% RSLogix 500 project C8014 TOPCOAT B 20170512 CBP.RSS, saved by version 8.30.00.16 %
PROJECT "C8014"    % processor: MicroLogix 1400; MAIN_PROG %

PROGRAM FILES
  LAD 2 "MAIN_PROG"  16 rungs
  LAD 3 "TCB ENTRY"  5 rungs
  LAD 4 "TCB TUNNEL"  44 rungs
  LAD 5 "REWORK"  13 rungs
  LAD 6 "COMMS"  3 rungs
  LAD 7   4 rungs
  LAD 8 "GATE FTA"  12 rungs
  LAD 9 "Z142-145"  23 rungs
  LAD 10 "TO_GLAZE"  15 rungs
  LAD 11 "FROM_GLAZE"  17 rungs
  LAD 12 "TO_BARN"  5 rungs
  LAD 13 "FRM_REPAIR"  5 rungs

DATA FILES
  O0 OUTPUT  9 elements
  I1 INPUT  12 elements
  S2 STATUS  66 elements
  B3 BINARY  40 elements
  T4 TIMER  54 elements
  C5 COUNTER  10 elements
  R6 CONTROL  1 elements
  N7 INTEGER  100 elements
  F8 FLOAT  1 elements
  ST9   21 elements
  RI10   5 elements
  MG11   4 elements

LADDER 2 "MAIN_PROG"
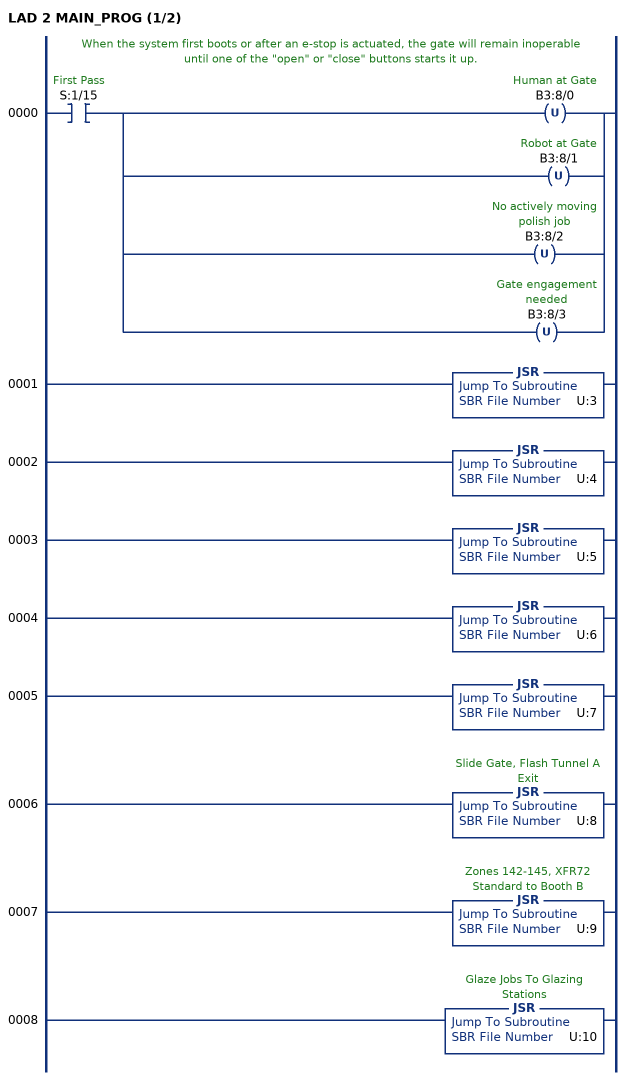
% Rung: 0 %
% When the system first boots or after an e-stop is actuated, the gate will remain inoperable until one of the "open" or "close" buttons starts it up. %
SOR XIC S:1/15 BST OTU B3:8/0 NXB OTU B3:8/1 NXB OTU B3:8/2 NXB OTU B3:8/3 BND EOR
%   S:1/15  "First Pass" %
%   B3:8/0  "Human at Gate" %
%   B3:8/1  "Robot at Gate" %
%   B3:8/2  "No actively moving polish job" %
%   B3:8/3  "Gate engagement needed" %
% Rung: 1 %
SOR JSR U:3 EOR
% Rung: 2 %
SOR JSR U:4 EOR
% Rung: 3 %
SOR JSR U:5 EOR
% Rung: 4 %
SOR JSR U:6 EOR
% Rung: 5 %
SOR JSR U:7 EOR
% Rung: 6 %
SOR JSR U:8 EOR
%   U:8  "Slide Gate, Flash Tunnel A Exit" %
% Rung: 7 %
SOR JSR U:9 EOR
%   U:9  "Zones 142-145, XFR72 Standard to Booth B" %
% Rung: 8 %
SOR JSR U:10 EOR
%   U:10  "Glaze Jobs To Glazing Stations" %

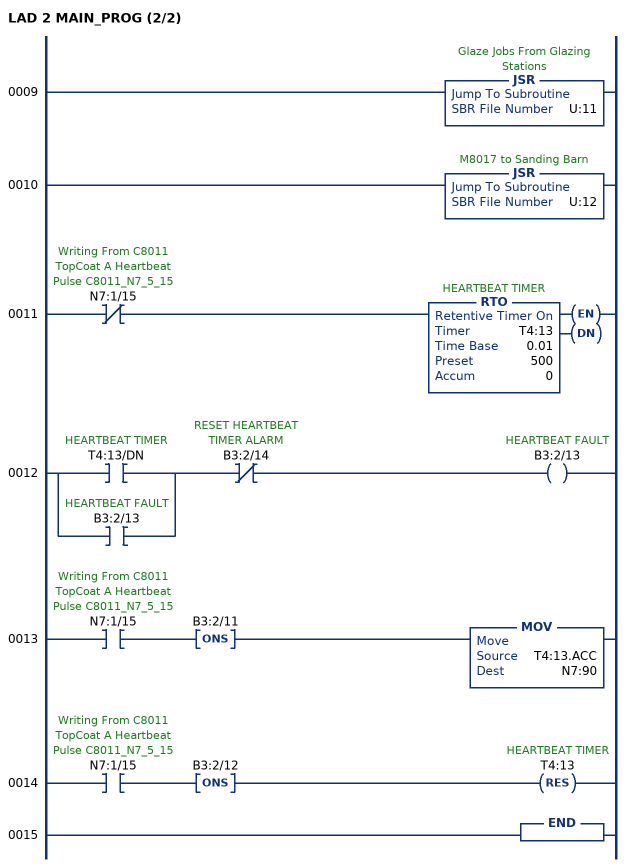
% Rung: 9 %
SOR JSR U:11 EOR
%   U:11  "Glaze Jobs From Glazing Stations" %
% Rung: 10 %
SOR JSR U:12 EOR
%   U:12  "M8017 to Sanding Barn" %
% Rung: 11 %
SOR XIO N7:1/15 RTO T4:13 0.01 500 0 EOR
%   N7:1/15  C8011_N7_5_15  "Writing From C8011 TopCoat A Heartbeat Pulse" %
%   T4:13  "HEARTBEAT TIMER" %
% Rung: 12 %
SOR BST XIC T4:13/DN NXB XIC B3:2/13 BND XIO B3:2/14 OTE B3:2/13 EOR
%   T4:13  "HEARTBEAT TIMER" %
%   B3:2/13  "HEARTBEAT FAULT" %
%   B3:2/14  "RESET HEARTBEAT TIMER ALARM" %
% Rung: 13 %
SOR XIC N7:1/15 ONS B3:2/11 MOV T4:13.ACC N7:90 EOR
%   N7:1/15  C8011_N7_5_15  "Writing From C8011 TopCoat A Heartbeat Pulse" %
%   T4:13  "HEARTBEAT TIMER" %
% Rung: 14 %
SOR XIC N7:1/15 ONS B3:2/12 RES T4:13 EOR
%   N7:1/15  C8011_N7_5_15  "Writing From C8011 TopCoat A Heartbeat Pulse" %
%   T4:13  "HEARTBEAT TIMER" %
% Rung: 15 %
SOR END EOR

LADDER 3 "TCB ENTRY"
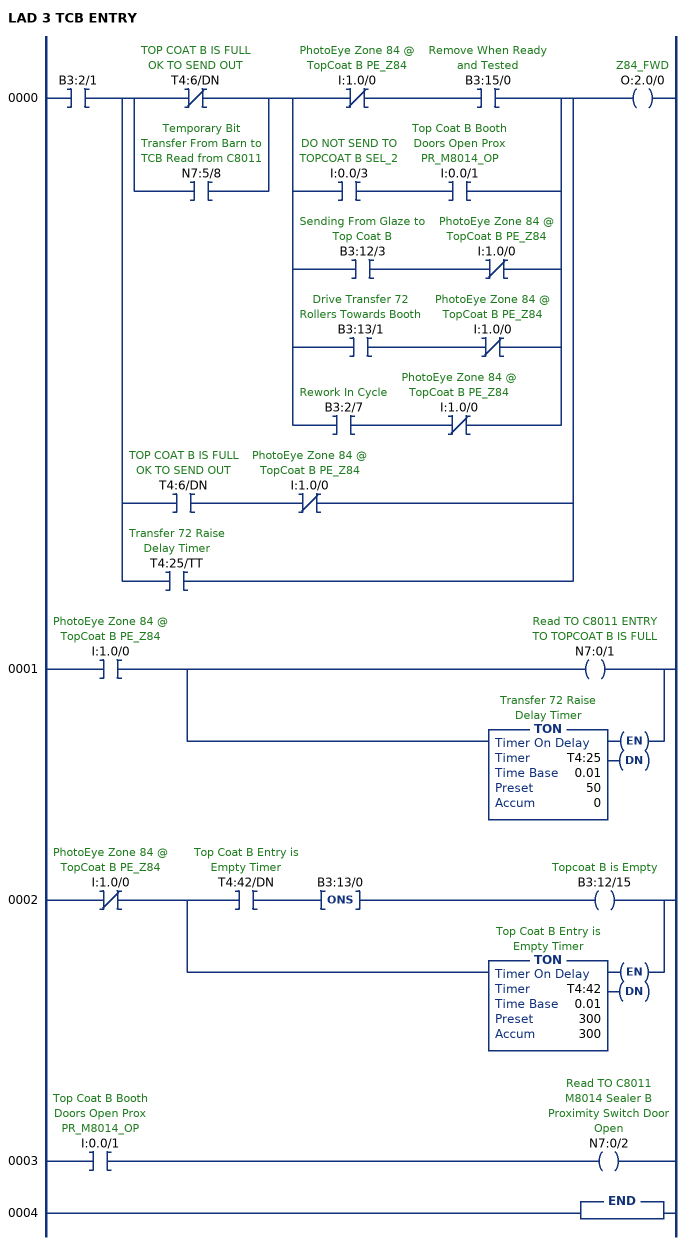
% Rung: 0 %
SOR XIC B3:2/1 BST BST XIO T4:6/DN NXB XIC N7:5/8 BND BST XIO I:1.0/0 XIC B3:15/0 NXB XIC I:0.0/3 XIC I:0.0/1 NXB XIC B3:12/3 XIO I:1.0/0 NXB XIC B3:13/1 XIO I:1.0/0 NXB XIC B3:2/7 XIO I:1.0/0 BND NXB XIC T4:6/DN XIO I:1.0/0 NXB XIC T4:25/TT BND OTE O:2.0/0 EOR
%   T4:6  "TOP COAT B IS FULL OK TO SEND OUT" %
%   N7:5/8  "Temporary Bit Transfer From Barn to TCB Read from C8011" %
%   I:1.0/0  PE_Z84  "PhotoEye Zone 84 @ TopCoat B" %
%   B3:15/0  "Remove When Ready and Tested" %
%   I:0.0/3  SEL_2  "DO NOT SEND TO TOPCOAT B" %
%   I:0.0/1  PR_M8014_OP  "Top Coat B Booth Doors Open Prox" %
%   B3:12/3  "Sending From Glaze to Top Coat B" %
%   B3:13/1  "Drive Transfer 72 Rollers Towards Booth" %
%   B3:2/7  "Rework In Cycle" %
%   T4:25  "Transfer 72 Raise Delay Timer" %
%   O:2.0/0  Z84_FWD %
% Rung: 1 %
SOR XIC I:1.0/0 BST OTE N7:0/1 NXB TON T4:25 0.01 50 0 BND EOR
%   I:1.0/0  PE_Z84  "PhotoEye Zone 84 @ TopCoat B" %
%   N7:0/1  "Read TO C8011 ENTRY TO TOPCOAT B IS FULL" %
%   T4:25  "Transfer 72 Raise Delay Timer" %
% Rung: 2 %
SOR XIO I:1.0/0 BST XIC T4:42/DN ONS B3:13/0 OTE B3:12/15 NXB TON T4:42 0.01 300 300 BND EOR
%   I:1.0/0  PE_Z84  "PhotoEye Zone 84 @ TopCoat B" %
%   T4:42  "Top Coat B Entry is Empty Timer" %
%   B3:12/15  "Topcoat B is Empty" %
% Rung: 3 %
SOR XIC I:0.0/1 OTE N7:0/2 EOR
%   I:0.0/1  PR_M8014_OP  "Top Coat B Booth Doors Open Prox" %
%   N7:0/2  "Read TO C8011 M8014 Sealer B Proximity Switch Door Open" %
% Rung: 4 %
SOR END EOR

LADDER 4 "TCB TUNNEL"
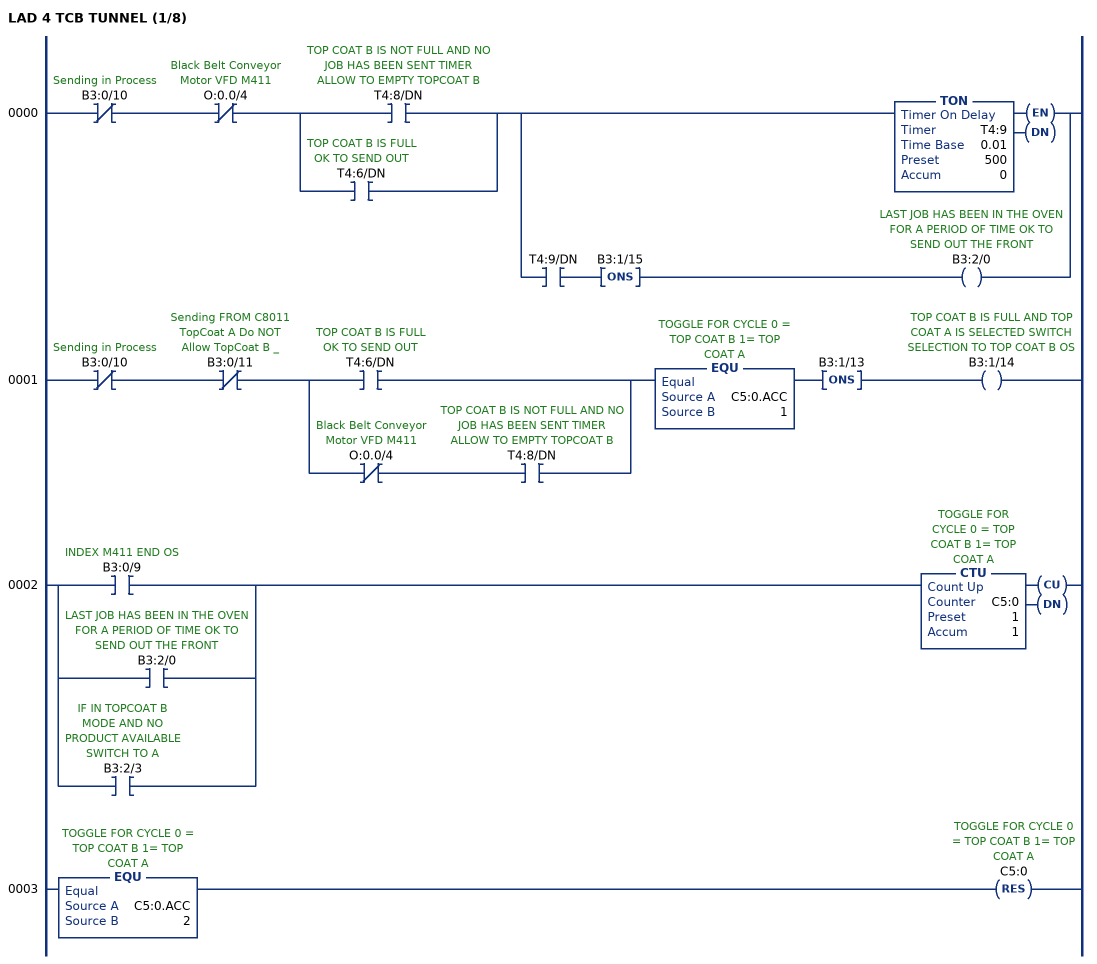
% Rung: 0 %
SOR XIO B3:0/10 XIO O:0.0/4 BST XIC T4:8/DN NXB XIC T4:6/DN BND BST TON T4:9 0.01 500 0 NXB XIC T4:9/DN ONS B3:1/15 OTE B3:2/0 BND EOR
%   B3:0/10  "Sending in Process" %
%   O:0.0/4  M411  "Black Belt Conveyor Motor VFD" %
%   T4:8  "TOP COAT B IS NOT FULL AND NO JOB HAS BEEN SENT TIMER ALLOW TO EMPTY TOPCOAT B" %
%   T4:6  "TOP COAT B IS FULL OK TO SEND OUT" %
%   B3:2/0  "LAST JOB HAS BEEN IN THE OVEN FOR A PERIOD OF TIME OK TO SEND OUT THE FRONT" %
% Rung: 1 %
SOR XIO B3:0/10 XIO B3:0/11 BST XIC T4:6/DN NXB XIO O:0.0/4 XIC T4:8/DN BND EQU C5:0.ACC 1 ONS B3:1/13 OTE B3:1/14 EOR
%   B3:0/10  "Sending in Process" %
%   B3:0/11  _  "Sending FROM C8011 TopCoat A Do NOT Allow TopCoat B" %
%   T4:6  "TOP COAT B IS FULL OK TO SEND OUT" %
%   O:0.0/4  M411  "Black Belt Conveyor Motor VFD" %
%   T4:8  "TOP COAT B IS NOT FULL AND NO JOB HAS BEEN SENT TIMER ALLOW TO EMPTY TOPCOAT B" %
%   C5:0  "TOGGLE FOR CYCLE 0 = TOP COAT B 1= TOP COAT A" %
%   B3:1/14  "TOP COAT B IS FULL AND TOP COAT A IS SELECTED SWITCH SELECTION TO TOP COAT B OS" %
% Rung: 2 %
SOR BST XIC B3:0/9 NXB XIC B3:2/0 NXB XIC B3:2/3 BND CTU C5:0 1 1 EOR
%   B3:0/9  "INDEX M411 END OS" %
%   B3:2/0  "LAST JOB HAS BEEN IN THE OVEN FOR A PERIOD OF TIME OK TO SEND OUT THE FRONT" %
%   B3:2/3  "IF IN TOPCOAT B MODE AND NO PRODUCT AVAILABLE SWITCH TO A" %
%   C5:0  "TOGGLE FOR CYCLE 0 = TOP COAT B 1= TOP COAT A" %
% Rung: 3 %
SOR EQU C5:0.ACC 2 RES C5:0 EOR
%   C5:0  "TOGGLE FOR CYCLE 0 = TOP COAT B 1= TOP COAT A" %

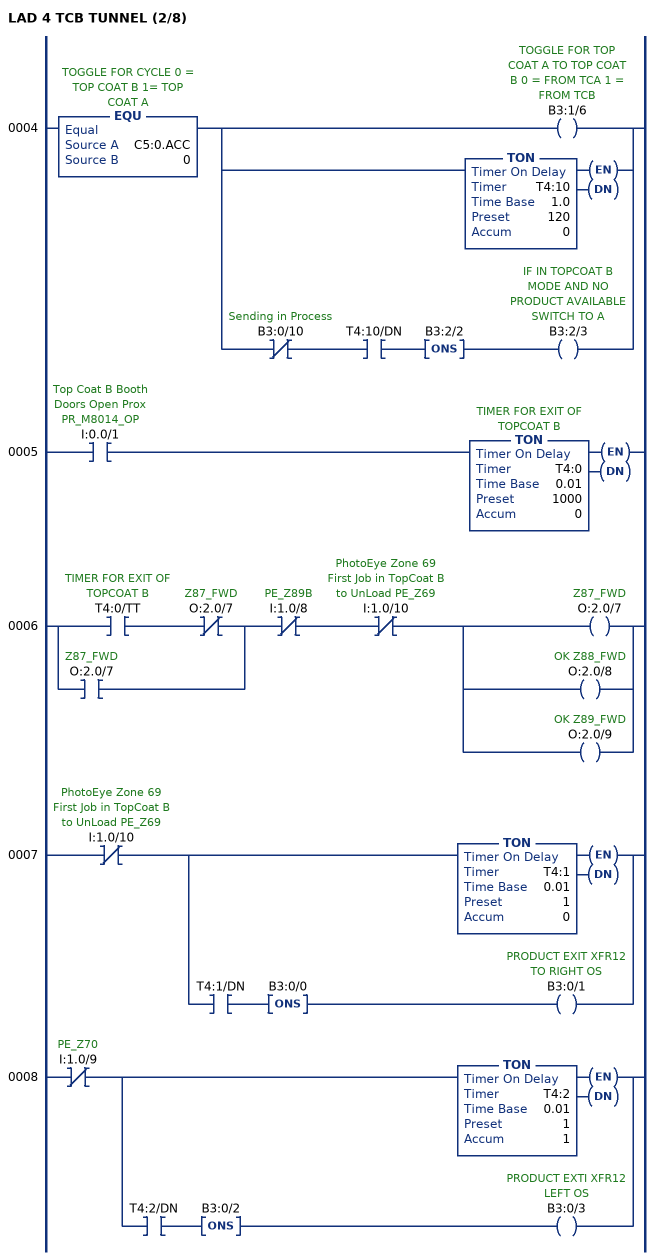
% Rung: 4 %
SOR EQU C5:0.ACC 0 BST OTE B3:1/6 NXB TON T4:10 1.0 120 0 NXB XIO B3:0/10 XIC T4:10/DN ONS B3:2/2 OTE B3:2/3 BND EOR
%   C5:0  "TOGGLE FOR CYCLE 0 = TOP COAT B 1= TOP COAT A" %
%   B3:1/6  "TOGGLE FOR TOP COAT A TO TOP COAT B 0 = FROM TCA 1 = FROM TCB" %
%   B3:0/10  "Sending in Process" %
%   B3:2/3  "IF IN TOPCOAT B MODE AND NO PRODUCT AVAILABLE SWITCH TO A" %
% Rung: 5 %
SOR XIC I:0.0/1 TON T4:0 0.01 1000 0 EOR
%   I:0.0/1  PR_M8014_OP  "Top Coat B Booth Doors Open Prox" %
%   T4:0  "TIMER FOR EXIT OF TOPCOAT B" %
% Rung: 6 %
SOR BST XIC T4:0/TT XIO O:2.0/7 NXB XIC O:2.0/7 BND XIO I:1.0/8 XIO I:1.0/10 BST OTE O:2.0/7 NXB OTE O:2.0/8 NXB OTE O:2.0/9 BND EOR
%   T4:0  "TIMER FOR EXIT OF TOPCOAT B" %
%   O:2.0/7  Z87_FWD %
%   I:1.0/8  PE_Z89B %
%   I:1.0/10  PE_Z69  "PhotoEye Zone 69 First Job in TopCoat B to UnLoad" %
%   O:2.0/8  Z88_FWD  "OK" %
%   O:2.0/9  Z89_FWD  "OK" %
% Rung: 7 %
SOR XIO I:1.0/10 BST TON T4:1 0.01 1 0 NXB XIC T4:1/DN ONS B3:0/0 OTE B3:0/1 BND EOR
%   I:1.0/10  PE_Z69  "PhotoEye Zone 69 First Job in TopCoat B to UnLoad" %
%   B3:0/1  "PRODUCT EXIT XFR12 TO RIGHT OS" %
% Rung: 8 %
SOR XIO I:1.0/9 BST TON T4:2 0.01 1 1 NXB XIC T4:2/DN ONS B3:0/2 OTE B3:0/3 BND EOR
%   I:1.0/9  PE_Z70 %
%   B3:0/3  "PRODUCT EXTI XFR12 LEFT OS" %

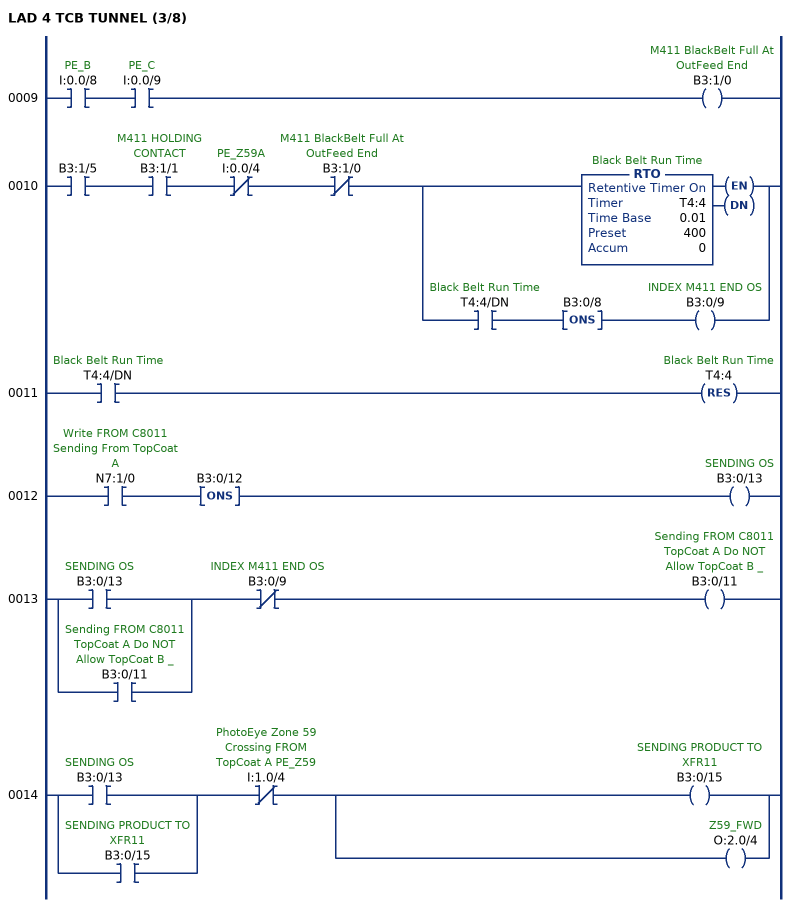
% Rung: 9 %
SOR XIC I:0.0/8 XIC I:0.0/9 OTE B3:1/0 EOR
%   I:0.0/8  PE_B %
%   I:0.0/9  PE_C %
%   B3:1/0  "M411 BlackBelt Full At OutFeed End" %
% Rung: 10 %
SOR XIC B3:1/5 XIC B3:1/1 XIO I:0.0/4 XIO B3:1/0 BST RTO T4:4 0.01 400 0 NXB XIC T4:4/DN ONS B3:0/8 OTE B3:0/9 BND EOR
%   B3:1/1  "M411 HOLDING CONTACT" %
%   I:0.0/4  PE_Z59A %
%   B3:1/0  "M411 BlackBelt Full At OutFeed End" %
%   T4:4  "Black Belt Run Time" %
%   B3:0/9  "INDEX M411 END OS" %
% Rung: 11 %
SOR XIC T4:4/DN RES T4:4 EOR
%   T4:4  "Black Belt Run Time" %
% Rung: 12 %
SOR XIC N7:1/0 ONS B3:0/12 OTE B3:0/13 EOR
%   N7:1/0  "Write FROM C8011 Sending From TopCoat A" %
%   B3:0/13  "SENDING OS" %
% Rung: 13 %
SOR BST XIC B3:0/13 NXB XIC B3:0/11 BND XIO B3:0/9 OTE B3:0/11 EOR
%   B3:0/13  "SENDING OS" %
%   B3:0/11  _  "Sending FROM C8011 TopCoat A Do NOT Allow TopCoat B" %
%   B3:0/9  "INDEX M411 END OS" %
% Rung: 14 %
SOR BST XIC B3:0/13 NXB XIC B3:0/15 BND XIO I:1.0/4 BST OTE B3:0/15 NXB OTE O:2.0/4 BND EOR
%   B3:0/13  "SENDING OS" %
%   B3:0/15  "SENDING PRODUCT TO XFR11" %
%   I:1.0/4  PE_Z59  "PhotoEye Zone 59 Crossing FROM TopCoat A" %
%   O:2.0/4  Z59_FWD %

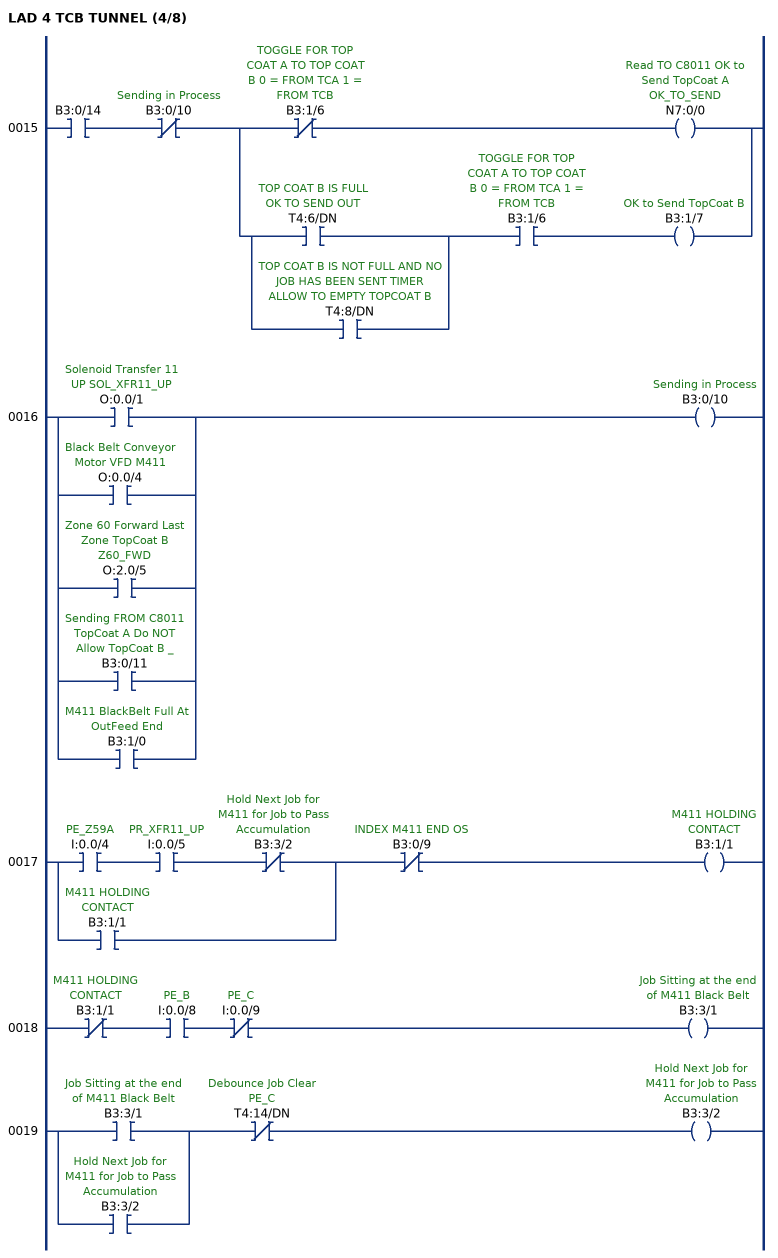
% Rung: 15 %
SOR XIC B3:0/14 XIO B3:0/10 BST XIO B3:1/6 OTE N7:0/0 NXB BST XIC T4:6/DN NXB XIC T4:8/DN BND XIC B3:1/6 OTE B3:1/7 BND EOR
%   B3:0/10  "Sending in Process" %
%   B3:1/6  "TOGGLE FOR TOP COAT A TO TOP COAT B 0 = FROM TCA 1 = FROM TCB" %
%   N7:0/0  OK_TO_SEND  "Read TO C8011 OK to Send TopCoat A" %
%   T4:6  "TOP COAT B IS FULL OK TO SEND OUT" %
%   T4:8  "TOP COAT B IS NOT FULL AND NO JOB HAS BEEN SENT TIMER ALLOW TO EMPTY TOPCOAT B" %
%   B3:1/7  "OK to Send TopCoat B" %
% Rung: 16 %
SOR BST XIC O:0.0/1 NXB XIC O:0.0/4 NXB XIC O:2.0/5 NXB XIC B3:0/11 NXB XIC B3:1/0 BND OTE B3:0/10 EOR
%   O:0.0/1  SOL_XFR11_UP  "Solenoid Transfer 11 UP" %
%   O:0.0/4  M411  "Black Belt Conveyor Motor VFD" %
%   O:2.0/5  Z60_FWD  "Zone 60 Forward Last Zone TopCoat B" %
%   B3:0/11  _  "Sending FROM C8011 TopCoat A Do NOT Allow TopCoat B" %
%   B3:1/0  "M411 BlackBelt Full At OutFeed End" %
%   B3:0/10  "Sending in Process" %
% Rung: 17 %
SOR BST XIC I:0.0/4 XIC I:0.0/5 XIO B3:3/2 NXB XIC B3:1/1 BND XIO B3:0/9 OTE B3:1/1 EOR
%   I:0.0/4  PE_Z59A %
%   I:0.0/5  PR_XFR11_UP %
%   B3:3/2  "Hold Next Job for M411 for Job to Pass Accumulation" %
%   B3:1/1  "M411 HOLDING CONTACT" %
%   B3:0/9  "INDEX M411 END OS" %
% Rung: 18 %
SOR XIO B3:1/1 XIC I:0.0/8 XIO I:0.0/9 OTE B3:3/1 EOR
%   B3:1/1  "M411 HOLDING CONTACT" %
%   I:0.0/8  PE_B %
%   I:0.0/9  PE_C %
%   B3:3/1  "Job Sitting at the end of M411 Black Belt" %
% Rung: 19 %
SOR BST XIC B3:3/1 NXB XIC B3:3/2 BND XIO T4:14/DN OTE B3:3/2 EOR
%   B3:3/1  "Job Sitting at the end of M411 Black Belt" %
%   B3:3/2  "Hold Next Job for M411 for Job to Pass Accumulation" %
%   T4:14  "Debounce Job Clear PE_C" %

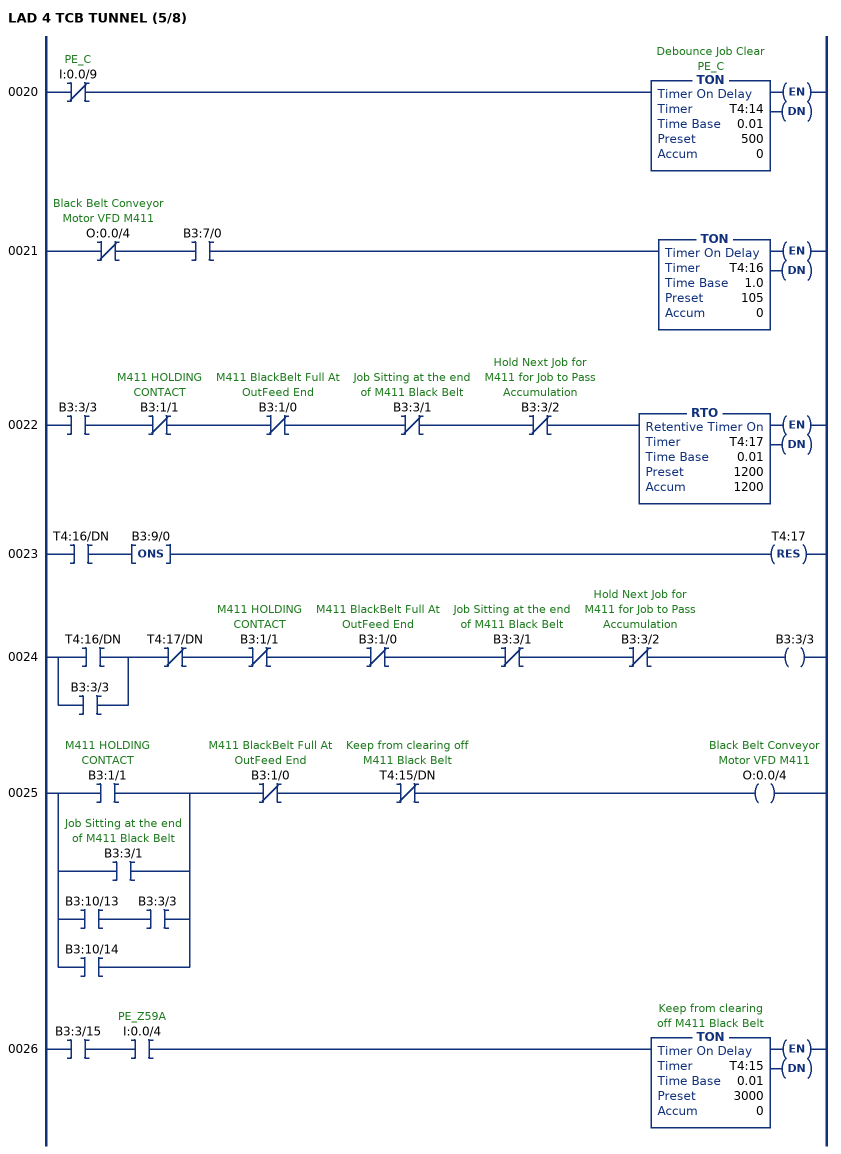
% Rung: 20 %
SOR XIO I:0.0/9 TON T4:14 0.01 500 0 EOR
%   I:0.0/9  PE_C %
%   T4:14  "Debounce Job Clear PE_C" %
% Rung: 21 %
SOR XIO O:0.0/4 XIC B3:7/0 TON T4:16 1.0 105 0 EOR
%   O:0.0/4  M411  "Black Belt Conveyor Motor VFD" %
% Rung: 22 %
SOR XIC B3:3/3 XIO B3:1/1 XIO B3:1/0 XIO B3:3/1 XIO B3:3/2 RTO T4:17 0.01 1200 1200 EOR
%   B3:1/1  "M411 HOLDING CONTACT" %
%   B3:1/0  "M411 BlackBelt Full At OutFeed End" %
%   B3:3/1  "Job Sitting at the end of M411 Black Belt" %
%   B3:3/2  "Hold Next Job for M411 for Job to Pass Accumulation" %
% Rung: 23 %
SOR XIC T4:16/DN ONS B3:9/0 RES T4:17 EOR
% Rung: 24 %
SOR BST XIC T4:16/DN NXB XIC B3:3/3 BND XIO T4:17/DN XIO B3:1/1 XIO B3:1/0 XIO B3:3/1 XIO B3:3/2 OTE B3:3/3 EOR
%   B3:1/1  "M411 HOLDING CONTACT" %
%   B3:1/0  "M411 BlackBelt Full At OutFeed End" %
%   B3:3/1  "Job Sitting at the end of M411 Black Belt" %
%   B3:3/2  "Hold Next Job for M411 for Job to Pass Accumulation" %
% Rung: 25 %
SOR BST XIC B3:1/1 NXB XIC B3:3/1 NXB XIC B3:10/13 XIC B3:3/3 NXB XIC B3:10/14 BND XIO B3:1/0 XIO T4:15/DN OTE O:0.0/4 EOR
%   B3:1/1  "M411 HOLDING CONTACT" %
%   B3:3/1  "Job Sitting at the end of M411 Black Belt" %
%   B3:1/0  "M411 BlackBelt Full At OutFeed End" %
%   T4:15  "Keep from clearing off M411 Black Belt" %
%   O:0.0/4  M411  "Black Belt Conveyor Motor VFD" %
% Rung: 26 %
SOR XIC B3:3/15 XIC I:0.0/4 TON T4:15 0.01 3000 0 EOR
%   I:0.0/4  PE_Z59A %
%   T4:15  "Keep from clearing off M411 Black Belt" %

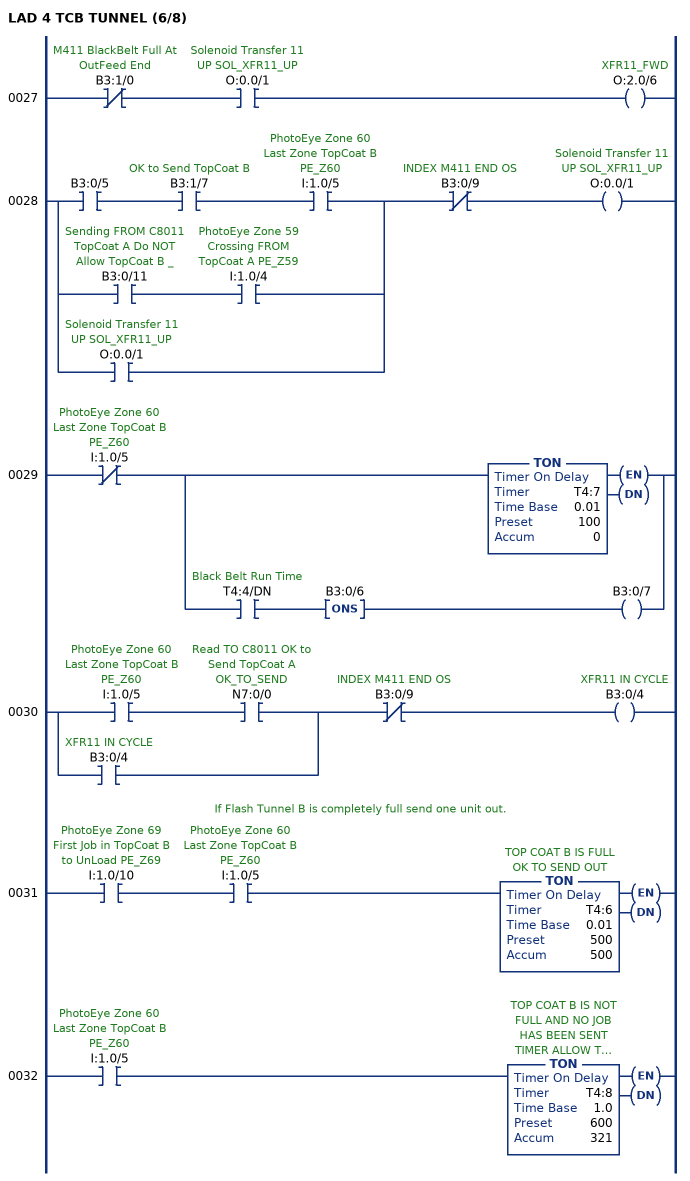
% Rung: 27 %
SOR XIO B3:1/0 XIC O:0.0/1 OTE O:2.0/6 EOR
%   B3:1/0  "M411 BlackBelt Full At OutFeed End" %
%   O:0.0/1  SOL_XFR11_UP  "Solenoid Transfer 11 UP" %
%   O:2.0/6  XFR11_FWD %
% Rung: 28 %
SOR BST BST XIC B3:0/5 XIC B3:1/7 XIC I:1.0/5 NXB XIC B3:0/11 XIC I:1.0/4 BND NXB XIC O:0.0/1 BND XIO B3:0/9 OTE O:0.0/1 EOR
%   B3:1/7  "OK to Send TopCoat B" %
%   I:1.0/5  PE_Z60  "PhotoEye Zone 60 Last Zone TopCoat B" %
%   B3:0/11  _  "Sending FROM C8011 TopCoat A Do NOT Allow TopCoat B" %
%   I:1.0/4  PE_Z59  "PhotoEye Zone 59 Crossing FROM TopCoat A" %
%   O:0.0/1  SOL_XFR11_UP  "Solenoid Transfer 11 UP" %
%   B3:0/9  "INDEX M411 END OS" %
% Rung: 29 %
SOR XIO I:1.0/5 BST TON T4:7 0.01 100 0 NXB XIC T4:4/DN ONS B3:0/6 OTE B3:0/7 BND EOR
%   I:1.0/5  PE_Z60  "PhotoEye Zone 60 Last Zone TopCoat B" %
%   T4:4  "Black Belt Run Time" %
% Rung: 30 %
SOR BST XIC I:1.0/5 XIC N7:0/0 NXB XIC B3:0/4 BND XIO B3:0/9 OTE B3:0/4 EOR
%   I:1.0/5  PE_Z60  "PhotoEye Zone 60 Last Zone TopCoat B" %
%   N7:0/0  OK_TO_SEND  "Read TO C8011 OK to Send TopCoat A" %
%   B3:0/4  "XFR11 IN CYCLE" %
%   B3:0/9  "INDEX M411 END OS" %
% Rung: 31 %
% If Flash Tunnel B is completely full send one unit out. %
SOR XIC I:1.0/10 XIC I:1.0/5 TON T4:6 0.01 500 500 EOR
%   I:1.0/10  PE_Z69  "PhotoEye Zone 69 First Job in TopCoat B to UnLoad" %
%   I:1.0/5  PE_Z60  "PhotoEye Zone 60 Last Zone TopCoat B" %
%   T4:6  "TOP COAT B IS FULL OK TO SEND OUT" %
% Rung: 32 %
SOR XIC I:1.0/5 TON T4:8 1.0 600 321 EOR
%   I:1.0/5  PE_Z60  "PhotoEye Zone 60 Last Zone TopCoat B" %
%   T4:8  "TOP COAT B IS NOT FULL AND NO JOB HAS BEEN SENT TIMER ALLOW TO EMPTY TOPCOAT B" %

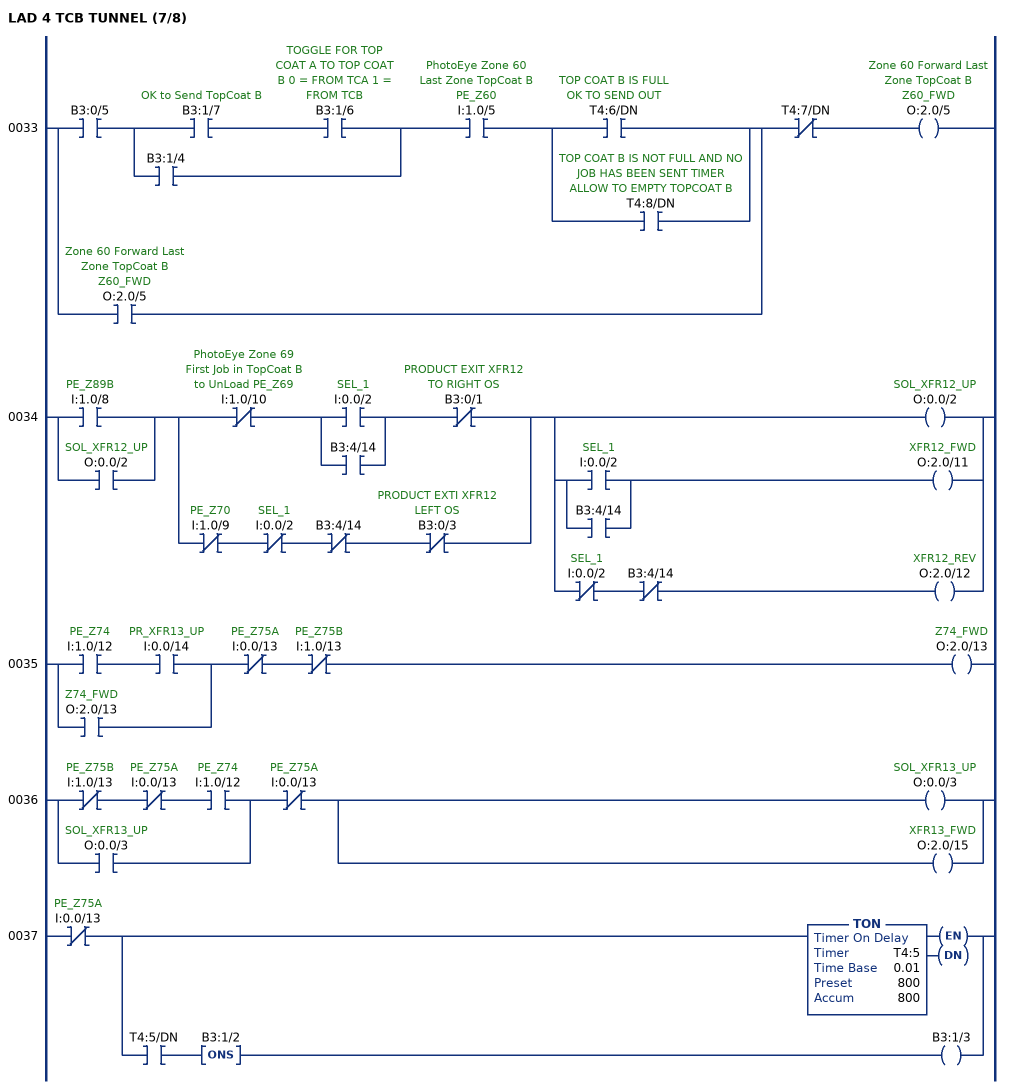
% Rung: 33 %
SOR BST XIC B3:0/5 BST XIC B3:1/7 XIC B3:1/6 NXB XIC B3:1/4 BND XIC I:1.0/5 BST XIC T4:6/DN NXB XIC T4:8/DN BND NXB XIC O:2.0/5 BND XIO T4:7/DN OTE O:2.0/5 EOR
%   B3:1/7  "OK to Send TopCoat B" %
%   B3:1/6  "TOGGLE FOR TOP COAT A TO TOP COAT B 0 = FROM TCA 1 = FROM TCB" %
%   I:1.0/5  PE_Z60  "PhotoEye Zone 60 Last Zone TopCoat B" %
%   T4:6  "TOP COAT B IS FULL OK TO SEND OUT" %
%   T4:8  "TOP COAT B IS NOT FULL AND NO JOB HAS BEEN SENT TIMER ALLOW TO EMPTY TOPCOAT B" %
%   O:2.0/5  Z60_FWD  "Zone 60 Forward Last Zone TopCoat B" %
% Rung: 34 %
SOR BST XIC I:1.0/8 NXB XIC O:0.0/2 BND BST XIO I:1.0/10 BST XIC I:0.0/2 NXB XIC B3:4/14 BND XIO B3:0/1 NXB XIO I:1.0/9 XIO I:0.0/2 XIO B3:4/14 XIO B3:0/3 BND BST OTE O:0.0/2 NXB BST XIC I:0.0/2 NXB XIC B3:4/14 BND OTE O:2.0/11 NXB XIO I:0.0/2 XIO B3:4/14 OTE O:2.0/12 BND EOR
%   I:1.0/8  PE_Z89B %
%   O:0.0/2  SOL_XFR12_UP %
%   I:1.0/10  PE_Z69  "PhotoEye Zone 69 First Job in TopCoat B to UnLoad" %
%   I:0.0/2  SEL_1 %
%   B3:0/1  "PRODUCT EXIT XFR12 TO RIGHT OS" %
%   I:1.0/9  PE_Z70 %
%   B3:0/3  "PRODUCT EXTI XFR12 LEFT OS" %
%   O:2.0/11  XFR12_FWD %
%   O:2.0/12  XFR12_REV %
% Rung: 35 %
SOR BST XIC I:1.0/12 XIC I:0.0/14 NXB XIC O:2.0/13 BND XIO I:0.0/13 XIO I:1.0/13 OTE O:2.0/13 EOR
%   I:1.0/12  PE_Z74 %
%   I:0.0/14  PR_XFR13_UP %
%   O:2.0/13  Z74_FWD %
%   I:0.0/13  PE_Z75A %
%   I:1.0/13  PE_Z75B %
% Rung: 36 %
SOR BST XIO I:1.0/13 XIO I:0.0/13 XIC I:1.0/12 NXB XIC O:0.0/3 BND XIO I:0.0/13 BST OTE O:0.0/3 NXB OTE O:2.0/15 BND EOR
%   I:1.0/13  PE_Z75B %
%   I:0.0/13  PE_Z75A %
%   I:1.0/12  PE_Z74 %
%   O:0.0/3  SOL_XFR13_UP %
%   O:2.0/15  XFR13_FWD %
% Rung: 37 %
SOR XIO I:0.0/13 BST TON T4:5 0.01 800 800 NXB XIC T4:5/DN ONS B3:1/2 OTE B3:1/3 BND EOR
%   I:0.0/13  PE_Z75A %

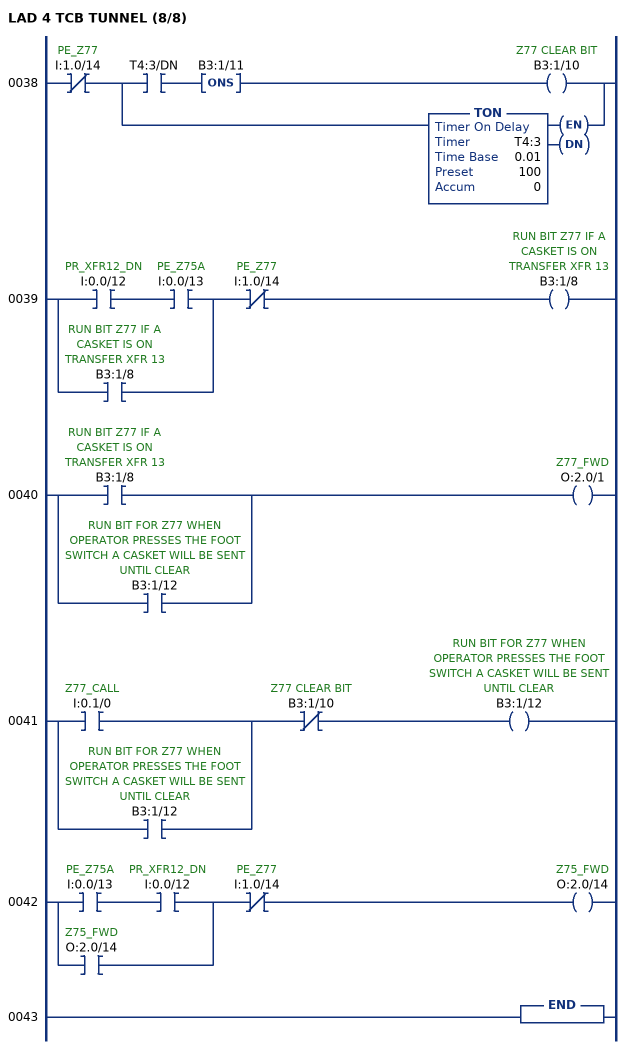
% Rung: 38 %
SOR XIO I:1.0/14 BST XIC T4:3/DN ONS B3:1/11 OTE B3:1/10 NXB TON T4:3 0.01 100 0 BND EOR
%   I:1.0/14  PE_Z77 %
%   B3:1/10  "Z77 CLEAR BIT" %
% Rung: 39 %
SOR BST XIC I:0.0/12 XIC I:0.0/13 NXB XIC B3:1/8 BND XIO I:1.0/14 OTE B3:1/8 EOR
%   I:0.0/12  PR_XFR12_DN %
%   I:0.0/13  PE_Z75A %
%   B3:1/8  "RUN BIT Z77 IF A CASKET IS ON TRANSFER XFR 13" %
%   I:1.0/14  PE_Z77 %
% Rung: 40 %
SOR BST XIC B3:1/8 NXB XIC B3:1/12 BND OTE O:2.0/1 EOR
%   B3:1/8  "RUN BIT Z77 IF A CASKET IS ON TRANSFER XFR 13" %
%   B3:1/12  "RUN BIT FOR Z77 WHEN OPERATOR PRESSES THE FOOT SWITCH A CASKET WILL BE SENT UNTIL CLEAR" %
%   O:2.0/1  Z77_FWD %
% Rung: 41 %
SOR BST XIC I:0.1/0 NXB XIC B3:1/12 BND XIO B3:1/10 OTE B3:1/12 EOR
%   I:0.1/0  Z77_CALL %
%   B3:1/12  "RUN BIT FOR Z77 WHEN OPERATOR PRESSES THE FOOT SWITCH A CASKET WILL BE SENT UNTIL CLEAR" %
%   B3:1/10  "Z77 CLEAR BIT" %
% Rung: 42 %
SOR BST XIC I:0.0/13 XIC I:0.0/12 NXB XIC O:2.0/14 BND XIO I:1.0/14 OTE O:2.0/14 EOR
%   I:0.0/13  PE_Z75A %
%   I:0.0/12  PR_XFR12_DN %
%   O:2.0/14  Z75_FWD %
%   I:1.0/14  PE_Z77 %
% Rung: 43 %
SOR END EOR

LADDER 5 "REWORK"
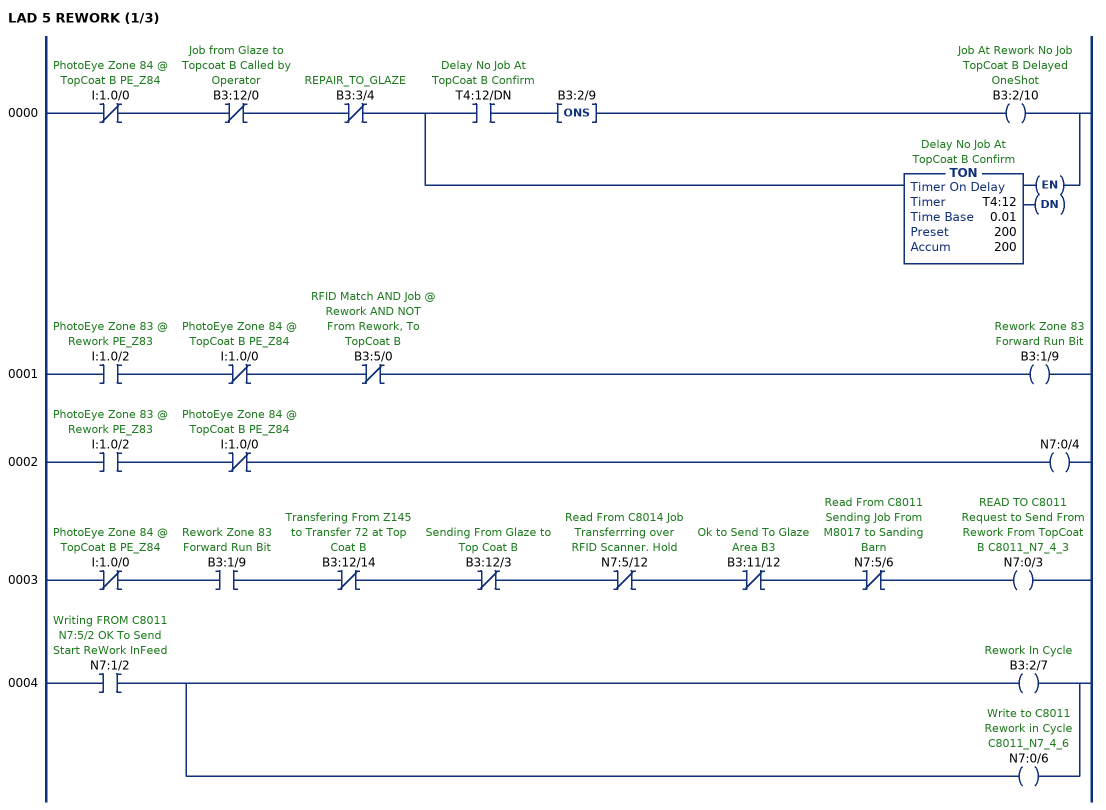
% Rung: 0 %
SOR XIO I:1.0/0 XIO B3:12/0 XIO B3:3/4 BST XIC T4:12/DN ONS B3:2/9 OTE B3:2/10 NXB TON T4:12 0.01 200 200 BND EOR
%   I:1.0/0  PE_Z84  "PhotoEye Zone 84 @ TopCoat B" %
%   B3:12/0  "Job from Glaze to Topcoat B Called by Operator" %
%   B3:3/4  REPAIR_TO_GLAZE %
%   T4:12  "Delay No Job At TopCoat B Confirm" %
%   B3:2/10  "Job At Rework No Job TopCoat B Delayed OneShot" %
% Rung: 1 %
SOR XIC I:1.0/2 XIO I:1.0/0 XIO B3:5/0 OTE B3:1/9 EOR
%   I:1.0/2  PE_Z83  "PhotoEye Zone 83 @ Rework" %
%   I:1.0/0  PE_Z84  "PhotoEye Zone 84 @ TopCoat B" %
%   B3:5/0  "RFID Match AND Job @ Rework AND NOT From Rework, To TopCoat B" %
%   B3:1/9  "Rework Zone 83 Forward Run Bit" %
% Rung: 2 %
SOR XIC I:1.0/2 XIO I:1.0/0 OTE N7:0/4 EOR
%   I:1.0/2  PE_Z83  "PhotoEye Zone 83 @ Rework" %
%   I:1.0/0  PE_Z84  "PhotoEye Zone 84 @ TopCoat B" %
% Rung: 3 %
SOR XIO I:1.0/0 XIC B3:1/9 XIO B3:12/14 XIO B3:12/3 XIO N7:5/12 XIO B3:11/12 XIO N7:5/6 OTE N7:0/3 EOR
%   I:1.0/0  PE_Z84  "PhotoEye Zone 84 @ TopCoat B" %
%   B3:1/9  "Rework Zone 83 Forward Run Bit" %
%   B3:12/14  "Transfering From Z145 to Transfer 72 at Top Coat B" %
%   B3:12/3  "Sending From Glaze to Top Coat B" %
%   N7:5/12  "Read From C8014 Job Transferrring over RFID Scanner. Hold" %
%   B3:11/12  B3  "Ok to Send To Glaze Area" %
%   N7:5/6  "Read From C8011 Sending Job From M8017 to Sanding Barn" %
%   N7:0/3  C8011_N7_4_3  "READ TO C8011 Request to Send From Rework From TopCoat B" %
% Rung: 4 %
SOR XIC N7:1/2 BST OTE B3:2/7 NXB OTE N7:0/6 BND EOR
%   N7:1/2  "Writing FROM C8011 N7:5/2 OK To Send Start ReWork InFeed" %
%   B3:2/7  "Rework In Cycle" %
%   N7:0/6  C8011_N7_4_6  "Write to C8011 Rework in Cycle" %

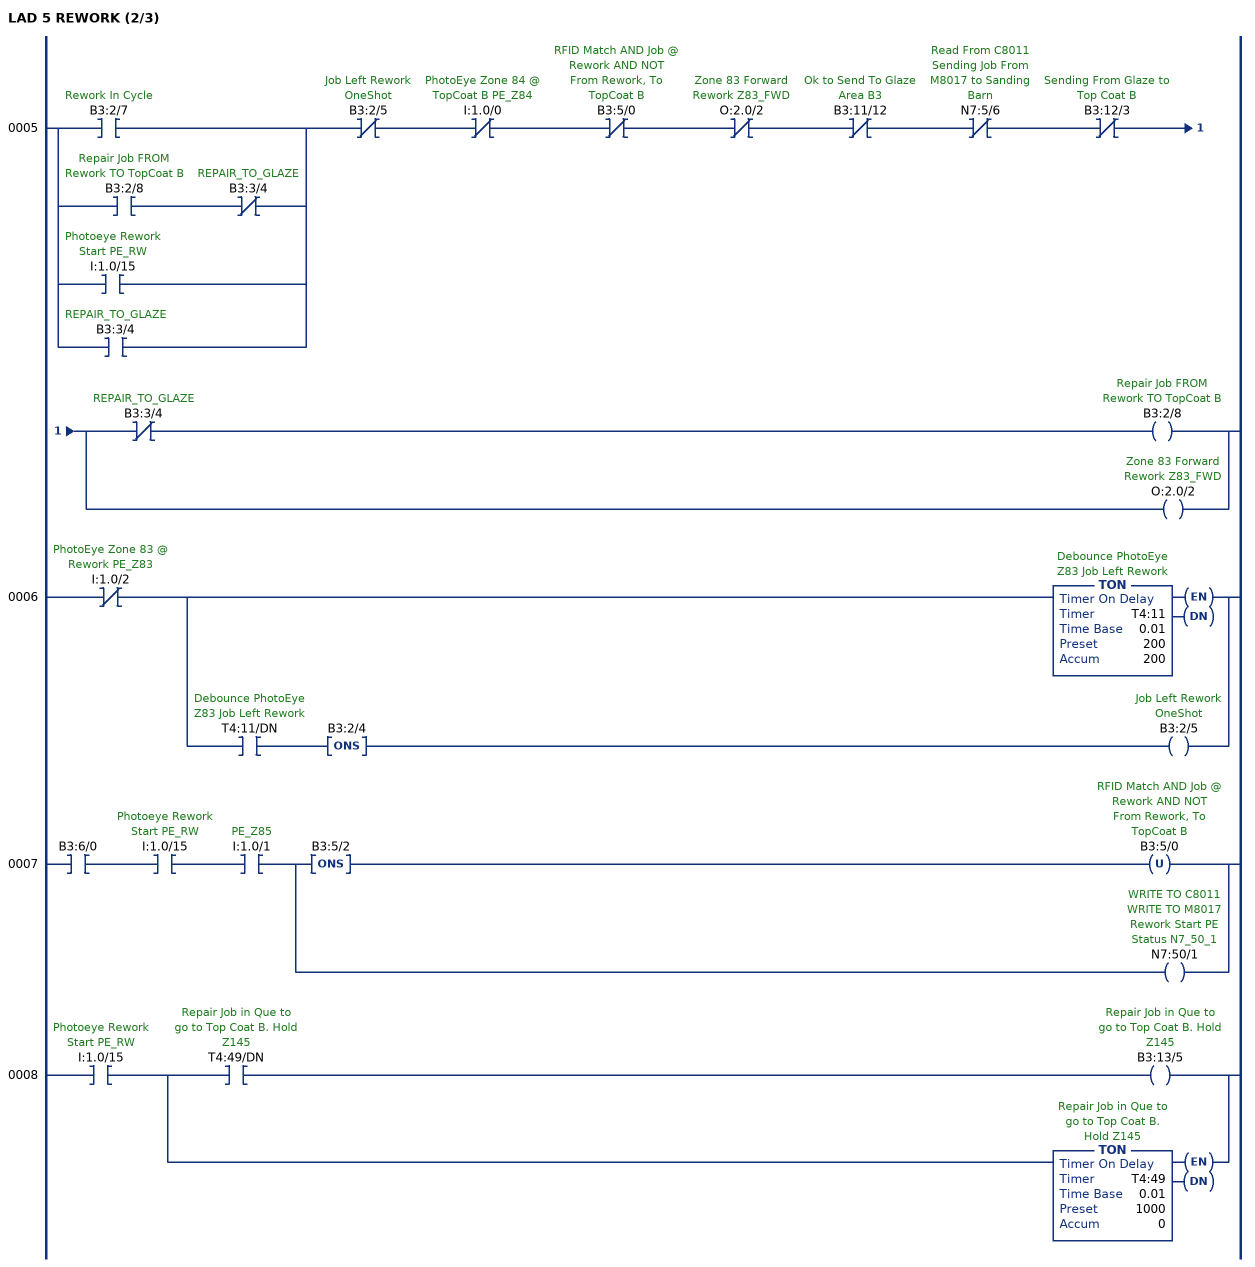
% Rung: 5 %
SOR BST XIC B3:2/7 NXB XIC B3:2/8 XIO B3:3/4 NXB XIC I:1.0/15 NXB XIC B3:3/4 BND XIO B3:2/5 XIO I:1.0/0 XIO B3:5/0 XIO O:2.0/2 XIO B3:11/12 XIO N7:5/6 XIO B3:12/3 BST XIO B3:3/4 OTE B3:2/8 NXB OTE O:2.0/2 BND EOR
%   B3:2/7  "Rework In Cycle" %
%   B3:2/8  "Repair Job FROM Rework TO TopCoat B" %
%   B3:3/4  REPAIR_TO_GLAZE %
%   I:1.0/15  PE_RW  "Photoeye Rework Start" %
%   B3:2/5  "Job Left Rework OneShot" %
%   I:1.0/0  PE_Z84  "PhotoEye Zone 84 @ TopCoat B" %
%   B3:5/0  "RFID Match AND Job @ Rework AND NOT From Rework, To TopCoat B" %
%   O:2.0/2  Z83_FWD  "Zone 83 Forward Rework" %
%   B3:11/12  B3  "Ok to Send To Glaze Area" %
%   N7:5/6  "Read From C8011 Sending Job From M8017 to Sanding Barn" %
%   B3:12/3  "Sending From Glaze to Top Coat B" %
% Rung: 6 %
SOR XIO I:1.0/2 BST TON T4:11 0.01 200 200 NXB XIC T4:11/DN ONS B3:2/4 OTE B3:2/5 BND EOR
%   I:1.0/2  PE_Z83  "PhotoEye Zone 83 @ Rework" %
%   T4:11  "Debounce PhotoEye Z83 Job Left Rework" %
%   B3:2/5  "Job Left Rework OneShot" %
% Rung: 7 %
SOR XIC B3:6/0 XIC I:1.0/15 XIC I:1.0/1 BST ONS B3:5/2 OTU B3:5/0 NXB OTE N7:50/1 BND EOR
%   I:1.0/15  PE_RW  "Photoeye Rework Start" %
%   I:1.0/1  PE_Z85 %
%   B3:5/0  "RFID Match AND Job @ Rework AND NOT From Rework, To TopCoat B" %
%   N7:50/1  N7_50_1  "WRITE TO C8011 WRITE TO M8017 Rework Start PE Status" %
% Rung: 8 %
SOR XIC I:1.0/15 BST XIC T4:49/DN OTE B3:13/5 NXB TON T4:49 0.01 1000 0 BND EOR
%   I:1.0/15  PE_RW  "Photoeye Rework Start" %
%   T4:49  "Repair Job in Que to go to Top Coat B. Hold Z145" %
%   B3:13/5  "Repair Job in Que to go to Top Coat B. Hold Z145" %

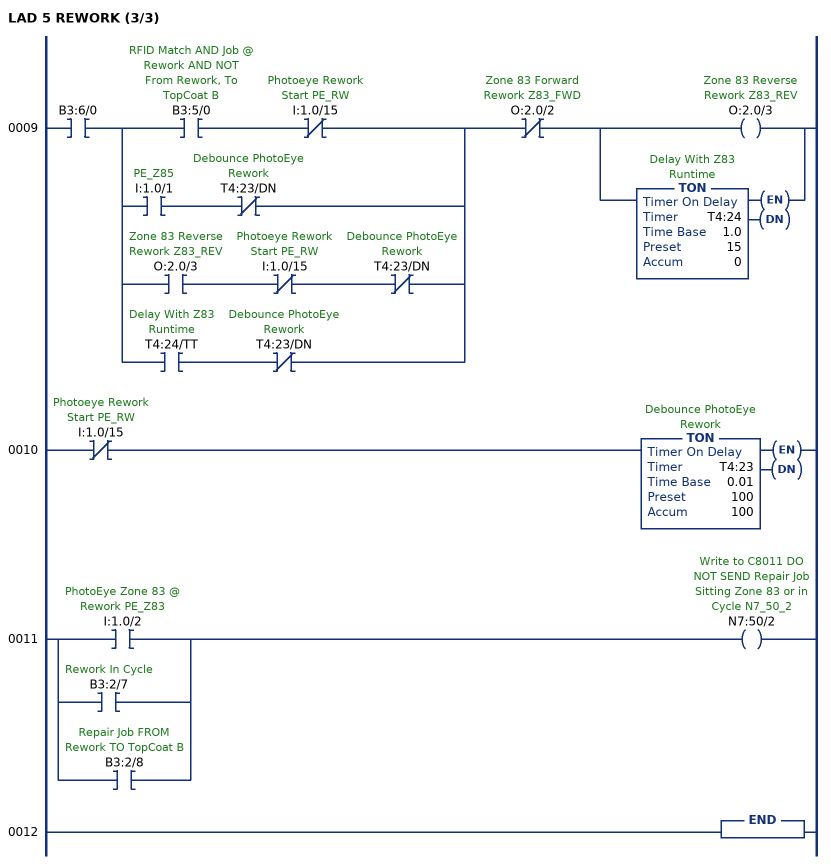
% Rung: 9 %
SOR XIC B3:6/0 BST XIC B3:5/0 XIO I:1.0/15 NXB XIC I:1.0/1 XIO T4:23/DN NXB XIC O:2.0/3 XIO I:1.0/15 XIO T4:23/DN NXB XIC T4:24/TT XIO T4:23/DN BND XIO O:2.0/2 BST OTE O:2.0/3 NXB TON T4:24 1.0 15 0 BND EOR
%   B3:5/0  "RFID Match AND Job @ Rework AND NOT From Rework, To TopCoat B" %
%   I:1.0/15  PE_RW  "Photoeye Rework Start" %
%   I:1.0/1  PE_Z85 %
%   T4:23  "Debounce PhotoEye Rework" %
%   O:2.0/3  Z83_REV  "Zone 83 Reverse Rework" %
%   T4:24  "Delay With Z83 Runtime" %
%   O:2.0/2  Z83_FWD  "Zone 83 Forward Rework" %
% Rung: 10 %
SOR XIO I:1.0/15 TON T4:23 0.01 100 100 EOR
%   I:1.0/15  PE_RW  "Photoeye Rework Start" %
%   T4:23  "Debounce PhotoEye Rework" %
% Rung: 11 %
SOR BST XIC I:1.0/2 NXB XIC B3:2/7 NXB XIC B3:2/8 BND OTE N7:50/2 EOR
%   I:1.0/2  PE_Z83  "PhotoEye Zone 83 @ Rework" %
%   B3:2/7  "Rework In Cycle" %
%   B3:2/8  "Repair Job FROM Rework TO TopCoat B" %
%   N7:50/2  N7_50_2  "Write to C8011 DO NOT SEND Repair Job Sitting Zone 83 or in Cycle" %
% Rung: 12 %
SOR END EOR

LADDER 6 "COMMS"
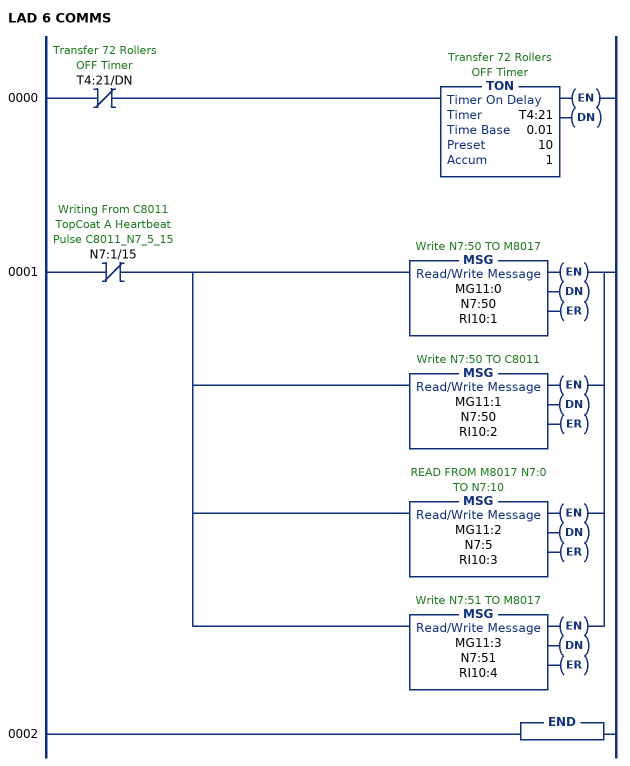
% Rung: 0 %
SOR XIO T4:21/DN TON T4:21 0.01 10 1 EOR
%   T4:21  "Transfer 72 Rollers OFF Timer" %
% Rung: 1 %
SOR XIO N7:1/15 BST MSG MG11:0 N7:50 RI10:1 NXB MSG MG11:1 N7:50 RI10:2 NXB MSG MG11:2 N7:5 RI10:3 NXB MSG MG11:3 N7:51 RI10:4 BND EOR
%   N7:1/15  C8011_N7_5_15  "Writing From C8011 TopCoat A Heartbeat Pulse" %
%   MSG set-up: 500CPU Write | 33 | 1 | N7:50 | N7:50 | 0 | 0 | 0 | 172.18.35.39 | 0 | 0 | 172.18.35.39 | RI10:1 %
%   MG11:0  "Write N7:50 TO M8017" %
%   MSG set-up: 500CPU Write | 33 | 1 | N7:50 | N7:50 | 0 | 0 | 0 | 172.18.35.32 | 0 | 0 | 172.18.35.32 | RI10:2 %
%   MG11:1  "Write N7:50 TO C8011" %
%   MSG set-up: 500CPU Read | 33 | 1 | N7:5 | N7:5 | 0 | 0 | 0 | 172.18.35.32 | 0 | 0 | 172.18.35.32 | RI10:3 %
%   MG11:2  "READ FROM M8017 N7:0 TO N7:10" %
%   MSG set-up: 500CPU Write | 5 | 1 | N7:51 | N7:51 | 0 | 0 | 0 | 172.18.35.39 | 0 | 0 | 172.18.35.39 | RI10:4 %
%   MG11:3  "Write N7:51 TO M8017" %
% Rung: 2 %
SOR END EOR

LADDER 7
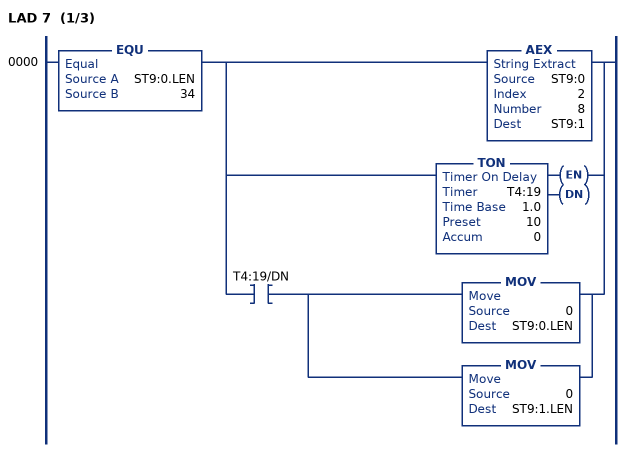
% Rung: 0 %
SOR EQU ST9:0.LEN 34 BST AEX ST9:0 2 8 ST9:1 NXB TON T4:19 1.0 10 0 NXB XIC T4:19/DN BST MOV 0 ST9:0.LEN NXB MOV 0 ST9:1.LEN BND BND EOR

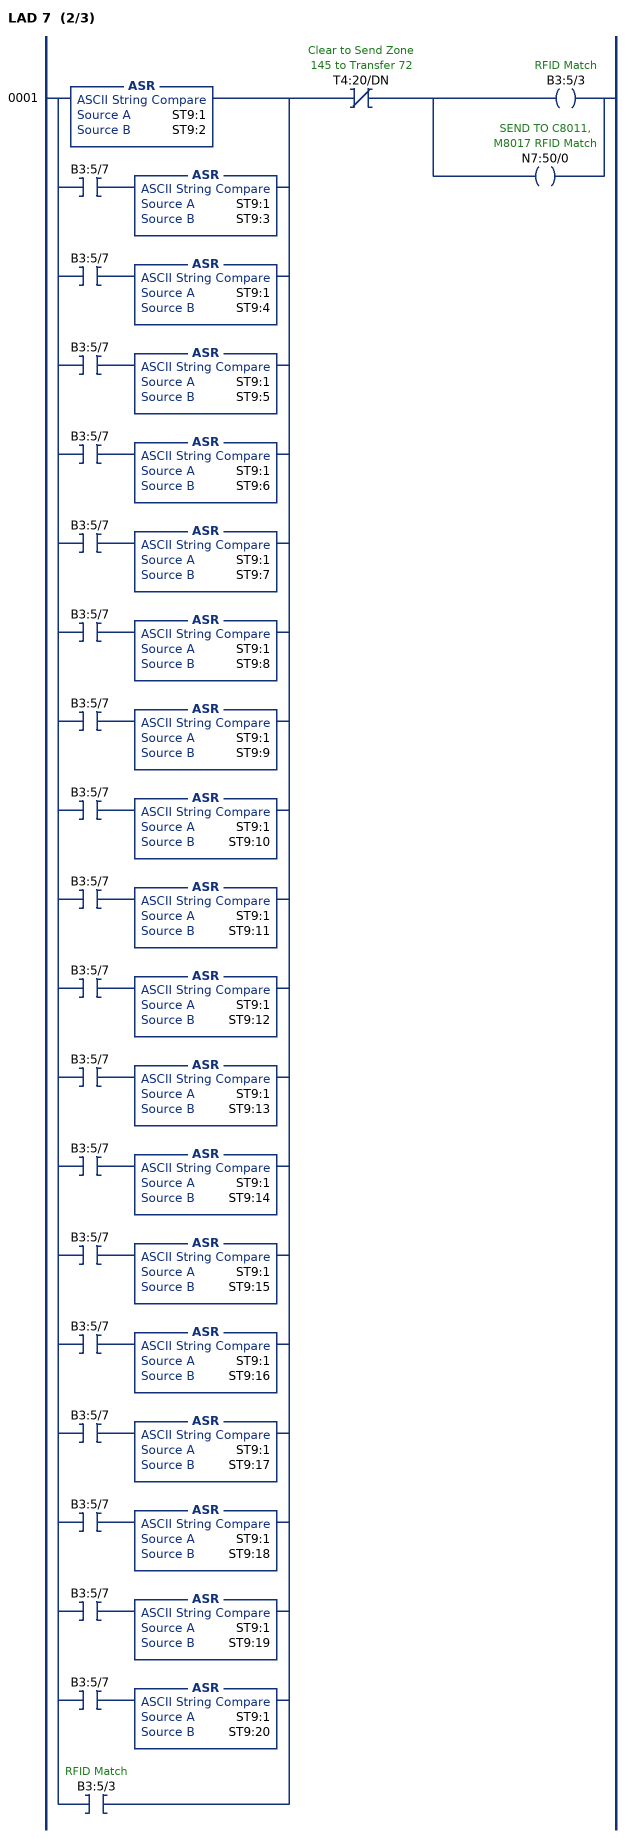
% Rung: 1 %
SOR BST ASR ST9:1 ST9:2 NXB XIC B3:5/7 ASR ST9:1 ST9:3 NXB XIC B3:5/7 ASR ST9:1 ST9:4 NXB XIC B3:5/7 ASR ST9:1 ST9:5 NXB XIC B3:5/7 ASR ST9:1 ST9:6 NXB XIC B3:5/7 ASR ST9:1 ST9:7 NXB XIC B3:5/7 ASR ST9:1 ST9:8 NXB XIC B3:5/7 ASR ST9:1 ST9:9 NXB XIC B3:5/7 ASR ST9:1 ST9:10 NXB XIC B3:5/7 ASR ST9:1 ST9:11 NXB XIC B3:5/7 ASR ST9:1 ST9:12 NXB XIC B3:5/7 ASR ST9:1 ST9:13 NXB XIC B3:5/7 ASR ST9:1 ST9:14 NXB XIC B3:5/7 ASR ST9:1 ST9:15 NXB XIC B3:5/7 ASR ST9:1 ST9:16 NXB XIC B3:5/7 ASR ST9:1 ST9:17 NXB XIC B3:5/7 ASR ST9:1 ST9:18 NXB XIC B3:5/7 ASR ST9:1 ST9:19 NXB XIC B3:5/7 ASR ST9:1 ST9:20 NXB XIC B3:5/3 BND XIO T4:20/DN BST OTE B3:5/3 NXB OTE N7:50/0 BND EOR
%   B3:5/3  "RFID Match" %
%   T4:20  "Clear to Send Zone 145 to Transfer 72" %
%   N7:50/0  "SEND TO C8011, M8017 RFID Match" %

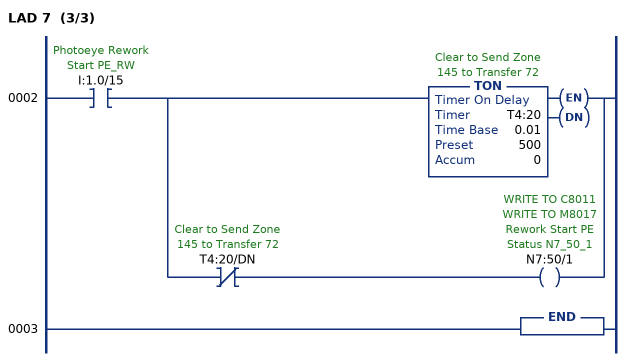
% Rung: 2 %
SOR XIC I:1.0/15 BST TON T4:20 0.01 500 0 NXB XIO T4:20/DN OTE N7:50/1 BND EOR
%   I:1.0/15  PE_RW  "Photoeye Rework Start" %
%   T4:20  "Clear to Send Zone 145 to Transfer 72" %
%   N7:50/1  N7_50_1  "WRITE TO C8011 WRITE TO M8017 Rework Start PE Status" %
% Rung: 3 %
SOR END EOR

LADDER 8 "GATE FTA"
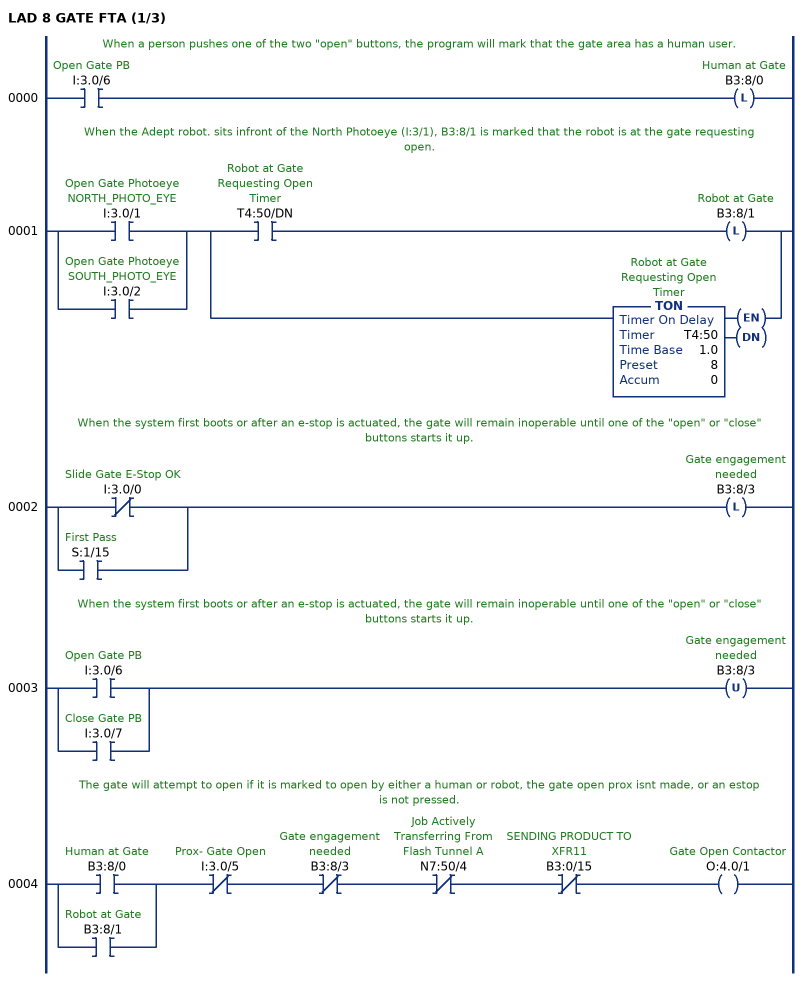
% Rung: 0 %
% When a person pushes one of the two "open" buttons, the program will mark that the gate area has a human user. %
SOR XIC I:3.0/6 OTL B3:8/0 EOR
%   I:3.0/6  "Open Gate PB" %
%   B3:8/0  "Human at Gate" %
% Rung: 1 %
% When the Adept robot. sits infront of the North Photoeye (I:3/1), B3:8/1 is marked that the robot is at the gate requesting open. %
SOR BST XIC I:3.0/1 NXB XIC I:3.0/2 BND BST XIC T4:50/DN OTL B3:8/1 NXB TON T4:50 1.0 8 0 BND EOR
%   I:3.0/1  NORTH_PHOTO_EYE  "Open Gate Photoeye" %
%   I:3.0/2  SOUTH_PHOTO_EYE  "Open Gate Photoeye" %
%   T4:50  "Robot at Gate Requesting Open Timer" %
%   B3:8/1  "Robot at Gate" %
% Rung: 2 %
% When the system first boots or after an e-stop is actuated, the gate will remain inoperable until one of the "open" or "close" buttons starts it up. %
SOR BST XIO I:3.0/0 NXB XIC S:1/15 BND OTL B3:8/3 EOR
%   I:3.0/0  "Slide Gate E-Stop OK" %
%   S:1/15  "First Pass" %
%   B3:8/3  "Gate engagement needed" %
% Rung: 3 %
% When the system first boots or after an e-stop is actuated, the gate will remain inoperable until one of the "open" or "close" buttons starts it up. %
SOR BST XIC I:3.0/6 NXB XIC I:3.0/7 BND OTU B3:8/3 EOR
%   I:3.0/6  "Open Gate PB" %
%   I:3.0/7  "Close Gate PB" %
%   B3:8/3  "Gate engagement needed" %
% Rung: 4 %
% The gate will attempt to open if it is marked to open by either a human or robot, the gate open prox isnt made, or an estop is not pressed. %
SOR BST XIC B3:8/0 NXB XIC B3:8/1 BND XIO I:3.0/5 XIO B3:8/3 XIO N7:50/4 XIO B3:0/15 OTE O:4.0/1 EOR
%   B3:8/0  "Human at Gate" %
%   B3:8/1  "Robot at Gate" %
%   I:3.0/5  "Prox- Gate Open" %
%   B3:8/3  "Gate engagement needed" %
%   N7:50/4  "Job Actively Transferring From Flash Tunnel A" %
%   B3:0/15  "SENDING PRODUCT TO XFR11" %
%   O:4.0/1  "Gate Open Contactor" %

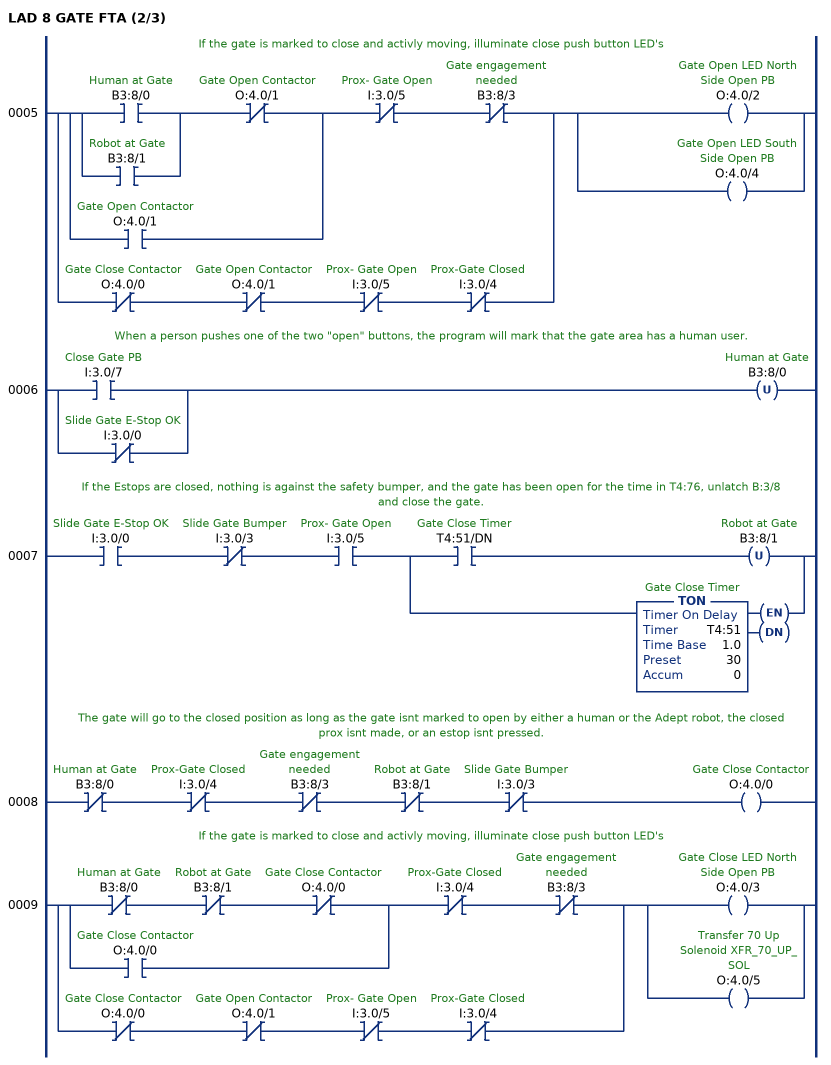
% Rung: 5 %
% If the gate is marked to close and activly moving, illuminate close push button LED's %
SOR BST BST BST XIC B3:8/0 NXB XIC B3:8/1 BND XIO O:4.0/1 NXB XIC O:4.0/1 BND XIO I:3.0/5 XIO B3:8/3 NXB XIO O:4.0/0 XIO O:4.0/1 XIO I:3.0/5 XIO I:3.0/4 BND BST OTE O:4.0/2 NXB OTE O:4.0/4 BND EOR
%   B3:8/0  "Human at Gate" %
%   B3:8/1  "Robot at Gate" %
%   O:4.0/1  "Gate Open Contactor" %
%   I:3.0/5  "Prox- Gate Open" %
%   B3:8/3  "Gate engagement needed" %
%   O:4.0/0  "Gate Close Contactor" %
%   I:3.0/4  "Prox-Gate Closed" %
%   O:4.0/2  "Gate Open LED North Side Open PB" %
%   O:4.0/4  "Gate Open LED South Side Open PB" %
% Rung: 6 %
% When a person pushes one of the two "open" buttons, the program will mark that the gate area has a human user. %
SOR BST XIC I:3.0/7 NXB XIO I:3.0/0 BND OTU B3:8/0 EOR
%   I:3.0/7  "Close Gate PB" %
%   I:3.0/0  "Slide Gate E-Stop OK" %
%   B3:8/0  "Human at Gate" %
% Rung: 7 %
% If the Estops are closed, nothing is against the safety bumper, and the gate has been open for the time in T4:76, unlatch B:3/8 and close the gate. %
SOR XIC I:3.0/0 XIO I:3.0/3 XIC I:3.0/5 BST XIC T4:51/DN OTU B3:8/1 NXB TON T4:51 1.0 30 0 BND EOR
%   I:3.0/0  "Slide Gate E-Stop OK" %
%   I:3.0/3  "Slide Gate Bumper" %
%   I:3.0/5  "Prox- Gate Open" %
%   T4:51  "Gate Close Timer" %
%   B3:8/1  "Robot at Gate" %
% Rung: 8 %
% The gate will go to the closed position as long as the gate isnt marked to open by either a human or the Adept robot, the closed prox isnt made, or an estop isnt pressed. %
SOR XIO B3:8/0 XIO I:3.0/4 XIO B3:8/3 XIO B3:8/1 XIO I:3.0/3 OTE O:4.0/0 EOR
%   B3:8/0  "Human at Gate" %
%   I:3.0/4  "Prox-Gate Closed" %
%   B3:8/3  "Gate engagement needed" %
%   B3:8/1  "Robot at Gate" %
%   I:3.0/3  "Slide Gate Bumper" %
%   O:4.0/0  "Gate Close Contactor" %
% Rung: 9 %
% If the gate is marked to close and activly moving, illuminate close push button LED's %
SOR BST BST XIO B3:8/0 XIO B3:8/1 XIO O:4.0/0 NXB XIC O:4.0/0 BND XIO I:3.0/4 XIO B3:8/3 NXB XIO O:4.0/0 XIO O:4.0/1 XIO I:3.0/5 XIO I:3.0/4 BND BST OTE O:4.0/3 NXB OTE O:4.0/5 BND EOR
%   B3:8/0  "Human at Gate" %
%   B3:8/1  "Robot at Gate" %
%   O:4.0/0  "Gate Close Contactor" %
%   I:3.0/4  "Prox-Gate Closed" %
%   B3:8/3  "Gate engagement needed" %
%   O:4.0/1  "Gate Open Contactor" %
%   I:3.0/5  "Prox- Gate Open" %
%   O:4.0/3  "Gate Close LED North Side Open PB" %
%   O:4.0/5  XFR_70_UP_SOL  "Transfer 70 Up Solenoid" %

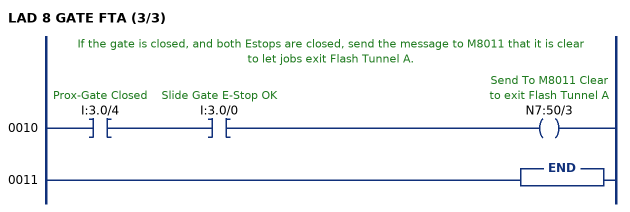
% Rung: 10 %
% If the gate is closed, and both Estops are closed, send the message to M8011 that it is clear to let jobs exit Flash Tunnel A. %
SOR XIC I:3.0/4 XIC I:3.0/0 OTE N7:50/3 EOR
%   I:3.0/4  "Prox-Gate Closed" %
%   I:3.0/0  "Slide Gate E-Stop OK" %
%   N7:50/3  "Send To M8011 Clear to exit Flash Tunnel A" %
% Rung: 11 %
SOR END EOR

LADDER 9 "Z142-145"
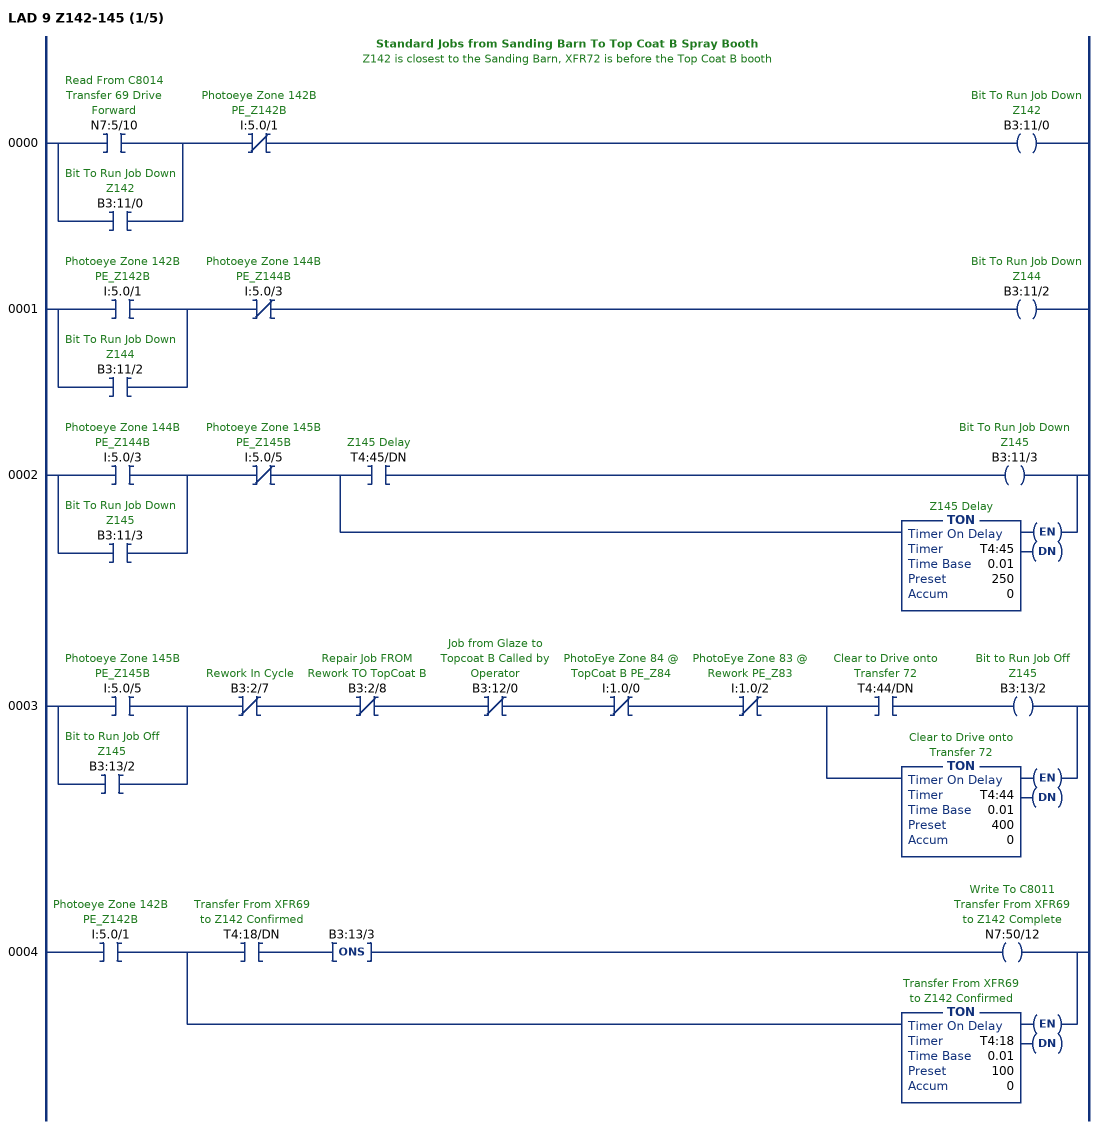
% Rung: 0 %
% TITLE: Standard Jobs from Sanding Barn To Top Coat B Spray Booth %
% Z142 is closest to the Sanding Barn, XFR72 is before the Top Coat B booth %
SOR BST XIC N7:5/10 NXB XIC B3:11/0 BND XIO I:5.0/1 OTE B3:11/0 EOR
%   N7:5/10  "Read From C8014 Transfer 69 Drive Forward" %
%   B3:11/0  "Bit To Run Job Down Z142" %
%   I:5.0/1  PE_Z142B  "Photoeye Zone 142B" %
% Rung: 1 %
SOR BST XIC I:5.0/1 NXB XIC B3:11/2 BND XIO I:5.0/3 OTE B3:11/2 EOR
%   I:5.0/1  PE_Z142B  "Photoeye Zone 142B" %
%   B3:11/2  "Bit To Run Job Down Z144" %
%   I:5.0/3  PE_Z144B  "Photoeye Zone 144B" %
% Rung: 2 %
SOR BST XIC I:5.0/3 NXB XIC B3:11/3 BND XIO I:5.0/5 BST XIC T4:45/DN OTE B3:11/3 NXB TON T4:45 0.01 250 0 BND EOR
%   I:5.0/3  PE_Z144B  "Photoeye Zone 144B" %
%   B3:11/3  "Bit To Run Job Down Z145" %
%   I:5.0/5  PE_Z145B  "Photoeye Zone 145B" %
%   T4:45  "Z145 Delay" %
% Rung: 3 %
SOR BST XIC I:5.0/5 NXB XIC B3:13/2 BND XIO B3:2/7 XIO B3:2/8 XIO B3:12/0 XIO I:1.0/0 XIO I:1.0/2 BST XIC T4:44/DN OTE B3:13/2 NXB TON T4:44 0.01 400 0 BND EOR
%   I:5.0/5  PE_Z145B  "Photoeye Zone 145B" %
%   B3:13/2  "Bit to Run Job Off Z145" %
%   B3:2/7  "Rework In Cycle" %
%   B3:2/8  "Repair Job FROM Rework TO TopCoat B" %
%   B3:12/0  "Job from Glaze to Topcoat B Called by Operator" %
%   I:1.0/0  PE_Z84  "PhotoEye Zone 84 @ TopCoat B" %
%   I:1.0/2  PE_Z83  "PhotoEye Zone 83 @ Rework" %
%   T4:44  "Clear to Drive onto Transfer 72" %
% Rung: 4 %
SOR XIC I:5.0/1 BST XIC T4:18/DN ONS B3:13/3 OTE N7:50/12 NXB TON T4:18 0.01 100 0 BND EOR
%   I:5.0/1  PE_Z142B  "Photoeye Zone 142B" %
%   T4:18  "Transfer From XFR69 to Z142 Confirmed" %
%   N7:50/12  "Write To C8011 Transfer From XFR69 to Z142 Complete" %

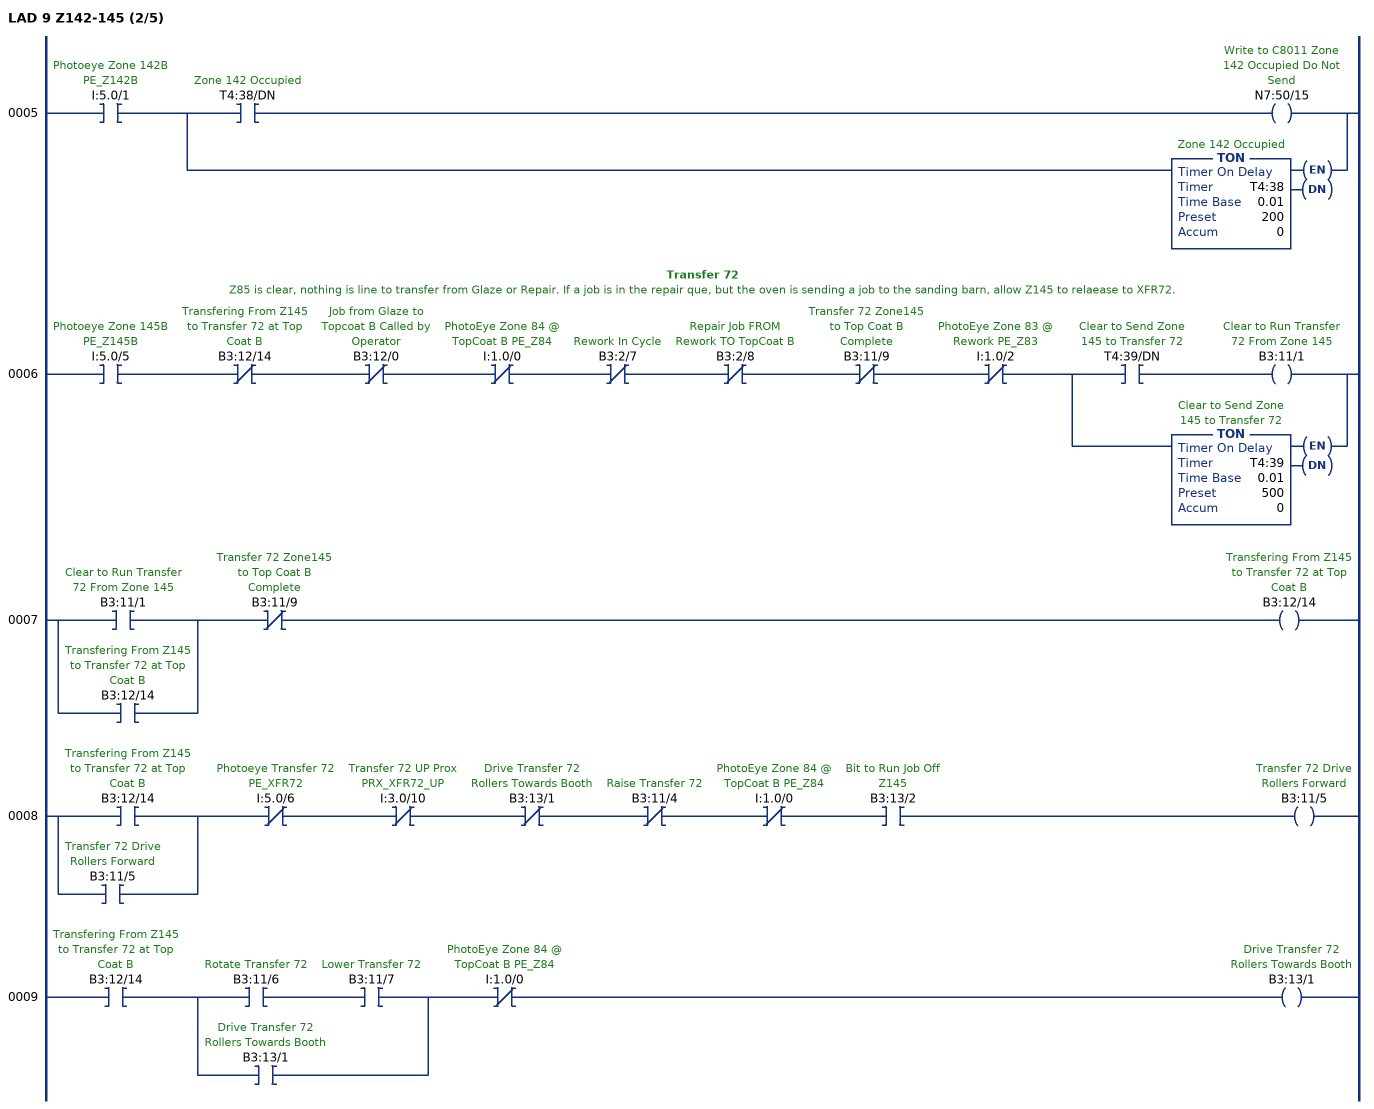
% Rung: 5 %
SOR XIC I:5.0/1 BST XIC T4:38/DN OTE N7:50/15 NXB TON T4:38 0.01 200 0 BND EOR
%   I:5.0/1  PE_Z142B  "Photoeye Zone 142B" %
%   T4:38  "Zone 142 Occupied" %
%   N7:50/15  "Write to C8011 Zone 142 Occupied Do Not Send" %
% Rung: 6 %
% TITLE: Transfer 72 %
% Z85 is clear, nothing is line to transfer from Glaze or Repair. If a job is in the repair que, but the oven is sending a job to the sanding barn, allow Z145 to relaease to XFR72. %
SOR XIC I:5.0/5 XIO B3:12/14 XIO B3:12/0 XIO I:1.0/0 XIO B3:2/7 XIO B3:2/8 XIO B3:11/9 XIO I:1.0/2 BST XIC T4:39/DN OTE B3:11/1 NXB TON T4:39 0.01 500 0 BND EOR
%   I:5.0/5  PE_Z145B  "Photoeye Zone 145B" %
%   B3:12/14  "Transfering From Z145 to Transfer 72 at Top Coat B" %
%   B3:12/0  "Job from Glaze to Topcoat B Called by Operator" %
%   I:1.0/0  PE_Z84  "PhotoEye Zone 84 @ TopCoat B" %
%   B3:2/7  "Rework In Cycle" %
%   B3:2/8  "Repair Job FROM Rework TO TopCoat B" %
%   B3:11/9  "Transfer 72 Zone145 to Top Coat B Complete" %
%   I:1.0/2  PE_Z83  "PhotoEye Zone 83 @ Rework" %
%   T4:39  "Clear to Send Zone 145 to Transfer 72" %
%   B3:11/1  "Clear to Run Transfer 72 From Zone 145" %
% Rung: 7 %
SOR BST XIC B3:11/1 NXB XIC B3:12/14 BND XIO B3:11/9 OTE B3:12/14 EOR
%   B3:11/1  "Clear to Run Transfer 72 From Zone 145" %
%   B3:12/14  "Transfering From Z145 to Transfer 72 at Top Coat B" %
%   B3:11/9  "Transfer 72 Zone145 to Top Coat B Complete" %
% Rung: 8 %
SOR BST XIC B3:12/14 NXB XIC B3:11/5 BND XIO I:5.0/6 XIO I:3.0/10 XIO B3:13/1 XIO B3:11/4 XIO I:1.0/0 XIC B3:13/2 OTE B3:11/5 EOR
%   B3:12/14  "Transfering From Z145 to Transfer 72 at Top Coat B" %
%   B3:11/5  "Transfer 72 Drive Rollers Forward" %
%   I:5.0/6  PE_XFR72  "Photoeye Transfer 72" %
%   I:3.0/10  PRX_XFR72_UP  "Transfer 72 UP Prox" %
%   B3:13/1  "Drive Transfer 72 Rollers Towards Booth" %
%   B3:11/4  "Raise Transfer 72" %
%   I:1.0/0  PE_Z84  "PhotoEye Zone 84 @ TopCoat B" %
%   B3:13/2  "Bit to Run Job Off Z145" %
% Rung: 9 %
SOR XIC B3:12/14 BST XIC B3:11/6 XIC B3:11/7 NXB XIC B3:13/1 BND XIO I:1.0/0 OTE B3:13/1 EOR
%   B3:12/14  "Transfering From Z145 to Transfer 72 at Top Coat B" %
%   B3:11/6  "Rotate Transfer 72" %
%   B3:11/7  "Lower Transfer 72" %
%   B3:13/1  "Drive Transfer 72 Rollers Towards Booth" %
%   I:1.0/0  PE_Z84  "PhotoEye Zone 84 @ TopCoat B" %

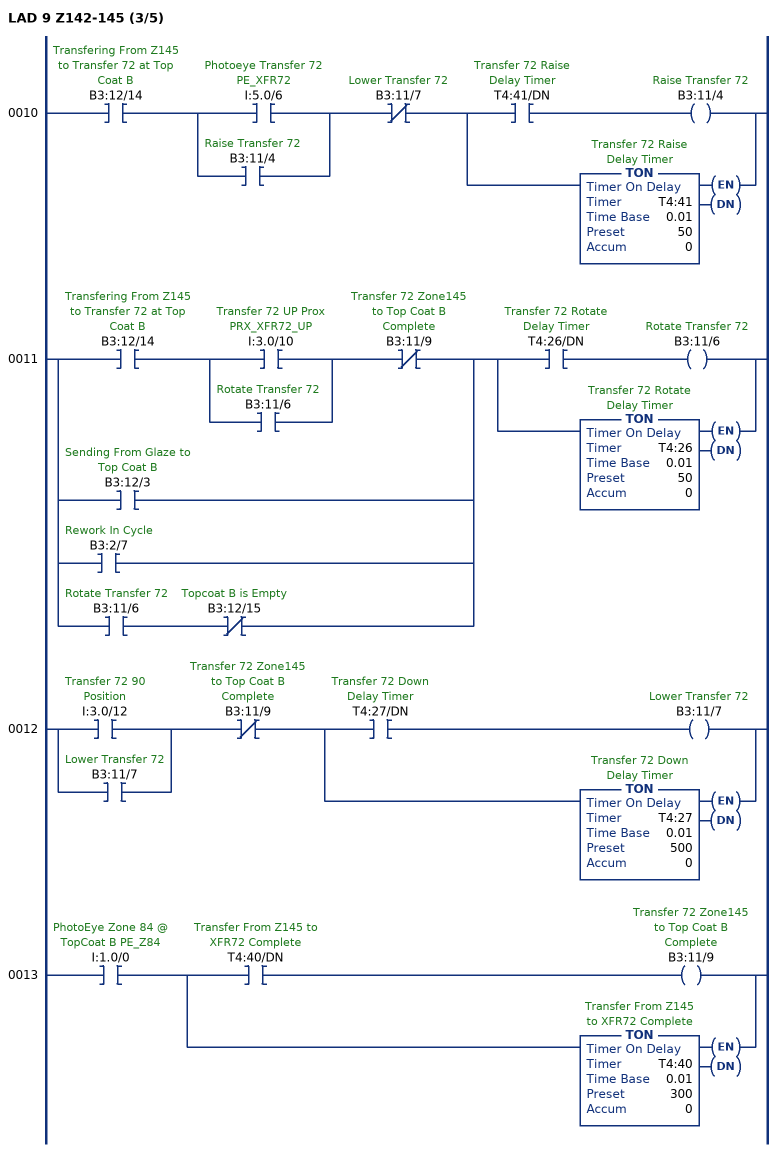
% Rung: 10 %
SOR XIC B3:12/14 BST XIC I:5.0/6 NXB XIC B3:11/4 BND XIO B3:11/7 BST XIC T4:41/DN OTE B3:11/4 NXB TON T4:41 0.01 50 0 BND EOR
%   B3:12/14  "Transfering From Z145 to Transfer 72 at Top Coat B" %
%   I:5.0/6  PE_XFR72  "Photoeye Transfer 72" %
%   B3:11/4  "Raise Transfer 72" %
%   B3:11/7  "Lower Transfer 72" %
%   T4:41  "Transfer 72 Raise Delay Timer" %
% Rung: 11 %
SOR BST XIC B3:12/14 BST XIC I:3.0/10 NXB XIC B3:11/6 BND XIO B3:11/9 NXB XIC B3:12/3 NXB XIC B3:2/7 NXB XIC B3:11/6 XIO B3:12/15 BND BST XIC T4:26/DN OTE B3:11/6 NXB TON T4:26 0.01 50 0 BND EOR
%   B3:12/14  "Transfering From Z145 to Transfer 72 at Top Coat B" %
%   I:3.0/10  PRX_XFR72_UP  "Transfer 72 UP Prox" %
%   B3:11/6  "Rotate Transfer 72" %
%   B3:11/9  "Transfer 72 Zone145 to Top Coat B Complete" %
%   B3:12/3  "Sending From Glaze to Top Coat B" %
%   B3:2/7  "Rework In Cycle" %
%   B3:12/15  "Topcoat B is Empty" %
%   T4:26  "Transfer 72 Rotate Delay Timer" %
% Rung: 12 %
SOR BST XIC I:3.0/12 NXB XIC B3:11/7 BND XIO B3:11/9 BST XIC T4:27/DN OTE B3:11/7 NXB TON T4:27 0.01 500 0 BND EOR
%   I:3.0/12  "Transfer 72 90 Position" %
%   B3:11/7  "Lower Transfer 72" %
%   B3:11/9  "Transfer 72 Zone145 to Top Coat B Complete" %
%   T4:27  "Transfer 72 Down Delay Timer" %
% Rung: 13 %
SOR XIC I:1.0/0 BST XIC T4:40/DN OTE B3:11/9 NXB TON T4:40 0.01 300 0 BND EOR
%   I:1.0/0  PE_Z84  "PhotoEye Zone 84 @ TopCoat B" %
%   T4:40  "Transfer From Z145 to XFR72 Complete" %
%   B3:11/9  "Transfer 72 Zone145 to Top Coat B Complete" %

